LIN {X 0,Y 579.705,Z 783.31,A -85,B 0,C 180,E1 8978.544,E2 8978.544} C_VEL
LIN {X 0,Y 579.773,Z 783.31,A -85,B 0,C 180,E1 8983.301,E2 8983.301} C_VEL
LIN {X 0,Y 579.9,Z 783.31,A -85,B 0,C 180,E1 8989.468,E2 8989.468} C_VEL
LIN {X 0,Y 580.075,Z 783.31,A -85,B 0,C 180,E1 8994.009,E2 8994.009} C_VEL
LIN {X 0,Y 580.176,Z 783.31,A -85,B 0,C 180,E1 8998.509,E2 8998.509} C_VEL
LIN {X 0,Y 580.153,Z 783.31,A -85,B 0,C 180,E1 9002.999,E2 9002.999} C_VEL
LIN {X 0,Y 580.034,Z 783.31,A -85,B 0,C 180,E1 9007.51,E2 9007.51} C_VEL
LIN {X 0,Y 579.911,Z 783.31,A -85,B 0,C 180,E1 9012.07,E2 9012.07} C_VEL
LIN {X 0,Y 579.778,Z 783.31,A -85,B 0,C 180,E1 9016.711,E2 9016.711} C_VEL
LIN {X 0,Y 579.644,Z 783.31,A -85,B 0,C 180,E1 9021.47,E2 9021.47} C_VEL
LIN {X 0,Y 579.509,Z 783.31,A -85,B 0,C 180,E1 9027.261,E2 9027.261} C_VEL
LIN {X 0,Y 579.423,Z 783.31,A -85,B 0,C 180,E1 9033.311,E2 9033.311} C_VEL
LIN {X 0,Y 579.308,Z 783.31,A -85,B 0,C 180,E1 9038.885,E2 9038.885} C_VEL
LIN {X 0,Y 579.314,Z 783.31,A -85,B 0,C 180,E1 9045.078,E2 9045.078} C_VEL
LIN {X 0,Y 579.261,Z 783.31,A -85,B 0,C 180,E1 9051.116,E2 9051.116} C_VEL
LIN {X 0,Y 579.338,Z 783.519,A -85,B 0,C 180,E1 9053.514,E2 9053.514} C_VEL
LIN {X 0,Y 586.271,Z 797.884,A -85,B 0,C 180,E1 9054.256,E2 9054.256} C_VEL
LIN {X 0,Y 606.499,Z 837.506,A -85,B 0,C 180,E1 9056.265,E2 9056.265} C_VEL
LIN {X 0,Y 604.839,Z 881.39,A -85,B 0,C 180,E1 9057.125,E2 9057.125} C_VEL
LIN {X 0,Y 601.624,Z 924.158,A -85,B 0,C 180,E1 9058.57,E2 9058.57} C_VEL
LIN {X 0,Y 597.504,Z 964.209,A -85,B 0,C 180,E1 9060.574,E2 9060.574} C_VEL
LIN {X 0,Y 592.954,Z 1002,A -85,B 0,C 180,E1 9063.195,E2 9063.195} C_VEL
LIN {X 0,Y 588.505,Z 1036.812,A -85,B 0,C 180,E1 9066.46,E2 9066.46} C_VEL
LIN {X 0,Y 585.021,Z 1066.221,A -85,B 0,C 180,E1 9070.129,E2 9070.129} C_VEL
LIN {X 0,Y 582.678,Z 1089.161,A -85,B 0,C 180,E1 9073.891,E2 9073.891} C_VEL
LIN {X 0,Y 581.268,Z 1107.45,A -85,B 0,C 180,E1 9077.965,E2 9077.965} C_VEL
LIN {X 0,Y 580.663,Z 1119.244,A -85,B 0,C 180,E1 9081.75,E2 9081.75} C_VEL
LIN {X 0,Y 580.435,Z 1126.566,A -85,B 0,C 180,E1 9085.51,E2 9085.51} C_VEL
LIN {X 0,Y 580.498,Z 1129.543,A -85,B 0,C 180,E1 9090.001,E2 9090.001} C_VEL
LIN {X 0,Y 580.468,Z 1126.438,A -85,B 0,C 180,E1 9094.493,E2 9094.493} C_VEL
LIN {X 0,Y 580.72,Z 1119.016,A -85,B 0,C 180,E1 9098.252,E2 9098.252} C_VEL
LIN {X 0,Y 581.35,Z 1105.632,A -85,B 0,C 180,E1 9102.406,E2 9102.406} C_VEL
LIN {X 0,Y 582.795,Z 1087.275,A -85,B 0,C 180,E1 9106.362,E2 9106.362} C_VEL
LIN {X 0,Y 585.372,Z 1062.818,A -85,B 0,C 180,E1 9110.256,E2 9110.256} C_VEL
LIN {X 0,Y 588.867,Z 1034.215,A -85,B 0,C 180,E1 9113.721,E2 9113.721} C_VEL
LIN {X 0,Y 592.925,Z 1002.541,A -85,B 0,C 180,E1 9116.67,E2 9116.67} C_VEL
LIN {X 0,Y 597.544,Z 964.371,A -85,B 0,C 180,E1 9119.322,E2 9119.322} C_VEL
LIN {X 0,Y 601.491,Z 925.349,A -85,B 0,C 180,E1 9121.289,E2 9121.289} C_VEL
LIN {X 0,Y 604.713,Z 881.532,A -85,B 0,C 180,E1 9122.788,E2 9122.788} C_VEL
LIN {X 0,Y 606.403,Z 837.307,A -85,B 0,C 180,E1 9123.653,E2 9123.653} C_VEL
LIN {X 0,Y 579.444,Z 784.213,A -85,B 0,C 180,E1 9126.374,E2 9126.374} C_VEL
LIN {X 0,Y 579.393,Z 783.31,A -85,B 0,C 180,E1 9126.442,E2 9126.442} C_VEL
LIN {X 0,Y 579.354,Z 783.31,A -85,B 0,C 180,E1 9130.832,E2 9130.832} C_VEL
LIN {X 0,Y 579.285,Z 783.31,A -85,B 0,C 180,E1 9137.086,E2 9137.086} C_VEL
LIN {X 0,Y 579.266,Z 783.31,A -85,B 0,C 180,E1 9143.012,E2 9143.012} C_VEL
LIN {X 0,Y 579.458,Z 783.31,A -85,B 0,C 180,E1 9148.466,E2 9148.466} C_VEL
LIN {X 0,Y 579.564,Z 783.31,A -85,B 0,C 180,E1 9153.609,E2 9153.609} C_VEL
LIN {X 0,Y 579.673,Z 783.31,A -85,B 0,C 180,E1 9158.531,E2 9158.531} C_VEL
LIN {X 0,Y 579.784,Z 783.31,A -85,B 0,C 180,E1 9163.289,E2 9163.289} C_VEL
LIN {X 0,Y 579.956,Z 783.31,A -85,B 0,C 180,E1 9169.458,E2 9169.458} C_VEL
LIN {X 0,Y 580.11,Z 783.31,A -85,B 0,C 180,E1 9173.998,E2 9173.998} C_VEL
LIN {X 0,Y 580.202,Z 783.31,A -85,B 0,C 180,E1 9178.498,E2 9178.498} C_VEL
LIN {X 0,Y 580.166,Z 783.31,A -85,B 0,C 180,E1 9182.988,E2 9182.988} C_VEL
LIN {X 0,Y 580.046,Z 783.31,A -85,B 0,C 180,E1 9187.498,E2 9187.498} C_VEL
LIN {X 0,Y 579.912,Z 783.31,A -85,B 0,C 180,E1 9192.058,E2 9192.058} C_VEL
LIN {X 0,Y 579.821,Z 783.31,A -85,B 0,C 180,E1 9196.698,E2 9196.698} C_VEL
LIN {X 0,Y 579.67,Z 783.31,A -85,B 0,C 180,E1 9201.457,E2 9201.457} C_VEL
LIN {X 0,Y 579.573,Z 783.31,A -85,B 0,C 180,E1 9207.268,E2 9207.268} C_VEL
LIN {X 0,Y 579.449,Z 783.31,A -85,B 0,C 180,E1 9213.296,E2 9213.296} C_VEL
LIN {X 0,Y 579.272,Z 783.31,A -85,B 0,C 180,E1 9218.873,E2 9218.873} C_VEL
LIN {X 0,Y 579.22,Z 783.31,A -85,B 0,C 180,E1 9225.065,E2 9225.065} C_VEL
LIN {X 0,Y 579.372,Z 784.035,A -85,B 0,C 180,E1 9230.209,E2 9230.209} C_VEL
LIN {X 0,Y 603.342,Z 834.228,A -85,B 0,C 180,E1 9232.711,E2 9232.711} C_VEL
LIN {X 0,Y 607.455,Z 844.899,A -85,B 0,C 180,E1 9233.167,E2 9233.167} C_VEL
LIN {X 0,Y 605.623,Z 880.743,A -85,B 0,C 180,E1 9233.925,E2 9233.925} C_VEL
LIN {X 0,Y 600.996,Z 897.494,A -85,B 0,C 180,E1 9234.191,E2 9234.191} C_VEL
LIN {X 0,Y 596.819,Z 911.913,A -85,B 0,C 180,E1 9234.489,E2 9234.489} C_VEL
LIN {X 0,Y 596.616,Z 913.947,A -85,B 0,C 180,E1 9234.563,E2 9234.563} C_VEL
LIN {X 0,Y 592.607,Z 957.43,A -85,B 0,C 180,E1 9236.508,E2 9236.508} C_VEL
LIN {X 0,Y 588.124,Z 997.916,A -85,B 0,C 180,E1 9238.984,E2 9238.984} C_VEL
LIN {X 0,Y 583.838,Z 1034.56,A -85,B 0,C 180,E1 9241.907,E2 9241.907} C_VEL
LIN {X 0,Y 579.934,Z 1067.538,A -85,B 0,C 180,E1 9245.289,E2 9245.289} C_VEL
LIN {X 0,Y 576.663,Z 1096.856,A -85,B 0,C 180,E1 9249.175,E2 9249.175} C_VEL
LIN {X 0,Y 574.483,Z 1120.889,A -85,B 0,C 180,E1 9253.389,E2 9253.389} C_VEL
LIN {X 0,Y 573.307,Z 1137.76,A -85,B 0,C 180,E1 9257.405,E2 9257.405} C_VEL
LIN {X 0,Y 572.746,Z 1150.067,A -85,B 0,C 180,E1 9261.633,E2 9261.633} C_VEL
LIN {X 0,Y 572.529,Z 1156.644,A -85,B 0,C 180,E1 9265.445,E2 9265.445} C_VEL
LIN {X 0,Y 572.546,Z 1159.5,A -85,B 0,C 180,E1 9269.999,E2 9269.999} C_VEL
LIN {X 0,Y 572.544,Z 1156.648,A -85,B 0,C 180,E1 9274.552,E2 9274.552} C_VEL
LIN {X 0,Y 572.681,Z 1150.072,A -85,B 0,C 180,E1 9278.366,E2 9278.366} C_VEL
LIN {X 0,Y 573.309,Z 1137.771,A -85,B 0,C 180,E1 9282.592,E2 9282.592} C_VEL
LIN {X 0,Y 574.508,Z 1120.878,A -85,B 0,C 180,E1 9286.611,E2 9286.611} C_VEL
LIN {X 0,Y 576.684,Z 1096.833,A -85,B 0,C 180,E1 9290.827,E2 9290.827} C_VEL
LIN {X 0,Y 579.978,Z 1067.55,A -85,B 0,C 180,E1 9294.706,E2 9294.706} C_VEL
LIN {X 0,Y 583.804,Z 1034.632,A -85,B 0,C 180,E1 9298.087,E2 9298.087} C_VEL
LIN {X 0,Y 588.083,Z 997.958,A -85,B 0,C 180,E1 9301.015,E2 9301.015} C_VEL
LIN {X 0,Y 592.561,Z 957.205,A -85,B 0,C 180,E1 9303.507,E2 9303.507} C_VEL
LIN {X 0,Y 596.709,Z 912.308,A -85,B 0,C 180,E1 9305.503,E2 9305.503} C_VEL
LIN {X 0,Y 599.983,Z 864.038,A -85,B 0,C 180,E1 9306.907,E2 9306.907} C_VEL
LIN {X 0,Y 600.287,Z 844.634,A -85,B 0,C 180,E1 9307.314,E2 9307.314} C_VEL
LIN {X 0,Y 578.673,Z 798.345,A -85,B 0,C 180,E1 9309.62,E2 9309.62} C_VEL
LIN {X 0,Y 571.585,Z 784.671,A -85,B 0,C 180,E1 9310.396,E2 9310.396} C_VEL
LIN {X 0,Y 571.457,Z 783.31,A -85,B 0,C 180,E1 9310.504,E2 9310.504} C_VEL
LIN {X 0,Y 571.362,Z 783.31,A -85,B 0,C 180,E1 9316.424,E2 9316.424} C_VEL
LIN {X 0,Y 571.447,Z 783.31,A -85,B 0,C 180,E1 9322.694,E2 9322.694} C_VEL
LIN {X 0,Y 571.538,Z 783.31,A -85,B 0,C 180,E1 9328.028,E2 9328.028} C_VEL
LIN {X 0,Y 571.694,Z 783.31,A -85,B 0,C 180,E1 9333.23,E2 9333.23} C_VEL
LIN {X 0,Y 571.764,Z 783.31,A -85,B 0,C 180,E1 9338.231,E2 9338.231} C_VEL
LIN {X 0,Y 571.84,Z 783.31,A -85,B 0,C 180,E1 9343.062,E2 9343.062} C_VEL
LIN {X 0,Y 571.945,Z 783.31,A -85,B 0,C 180,E1 9348.567,E2 9348.567} C_VEL
LIN {X 0,Y 572.179,Z 783.31,A -85,B 0,C 180,E1 9353.926,E2 9353.926} C_VEL
LIN {X 0,Y 572.274,Z 783.31,A -85,B 0,C 180,E1 9358.489,E2 9358.489} C_VEL
LIN {X 0,Y 572.253,Z 783.31,A -85,B 0,C 180,E1 9363.041,E2 9363.041} C_VEL
LIN {X 0,Y 572.117,Z 783.31,A -85,B 0,C 180,E1 9367.614,E2 9367.614} C_VEL
LIN {X 0,Y 572.013,Z 783.31,A -85,B 0,C 180,E1 9372.239,E2 9372.239} C_VEL
LIN {X 0,Y 571.803,Z 783.31,A -85,B 0,C 180,E1 9377.464,E2 9377.464} C_VEL
LIN {X 0,Y 571.684,Z 783.31,A -85,B 0,C 180,E1 9383.429,E2 9383.429} C_VEL
LIN {X 0,Y 571.542,Z 783.31,A -85,B 0,C 180,E1 9388.978,E2 9388.978} C_VEL
LIN {X 0,Y 571.413,Z 783.31,A -85,B 0,C 180,E1 9394.717,E2 9394.717} C_VEL
LIN {X 0,Y 571.347,Z 783.31,A -85,B 0,C 180,E1 9399.733,E2 9399.733} C_VEL
LIN {X 0,Y 571.329,Z 783.31,A -85,B 0,C 180,E1 9405.731,E2 9405.731} C_VEL
LIN {X 0,Y 571.304,Z 783.31,A -85,B 0,C 180,E1 9410.47,E2 9410.47} C_VEL
LIN {X 0,Y 571.377,Z 783.363,A -85,B 0,C 180,E1 9412.878,E2 9412.878} C_VEL
LIN {X 0,Y 575.876,Z 793.256,A -85,B 0,C 180,E1 9413.386,E2 9413.386} C_VEL
LIN {X 0,Y 599.985,Z 840.052,A -85,B 0,C 180,E1 9415.857,E2 9415.857} C_VEL
LIN {X 0,Y 598.239,Z 883.352,A -85,B 0,C 180,E1 9416.746,E2 9416.746} C_VEL
LIN {X 0,Y 594.976,Z 924.317,A -85,B 0,C 180,E1 9418.148,E2 9418.148} C_VEL
LIN {X 0,Y 590.642,Z 964.871,A -85,B 0,C 180,E1 9420.198,E2 9420.198} C_VEL
LIN {X 0,Y 585.854,Z 1002.667,A -85,B 0,C 180,E1 9422.847,E2 9422.847} C_VEL
LIN {X 0,Y 581.235,Z 1037.328,A -85,B 0,C 180,E1 9426.134,E2 9426.134} C_VEL
LIN {X 0,Y 577.487,Z 1066.722,A -85,B 0,C 180,E1 9429.858,E2 9429.858} C_VEL
LIN {X 0,Y 574.912,Z 1090.243,A -85,B 0,C 180,E1 9433.81,E2 9433.81} C_VEL
LIN {X 0,Y 573.435,Z 1108.002,A -85,B 0,C 180,E1 9437.862,E2 9437.862} C_VEL
LIN {X 0,Y 572.791,Z 1119.491,A -85,B 0,C 180,E1 9441.636,E2 9441.636} C_VEL
LIN {X 0,Y 572.549,Z 1126.783,A -85,B 0,C 180,E1 9445.448,E2 9445.448} C_VEL
LIN {X 0,Y 572.624,Z 1129.751,A -85,B 0,C 180,E1 9450.001,E2 9450.001} C_VEL
LIN {X 0,Y 572.577,Z 1126.658,A -85,B 0,C 180,E1 9454.555,E2 9454.555} C_VEL
LIN {X 0,Y 572.836,Z 1119.262,A -85,B 0,C 180,E1 9458.366,E2 9458.366} C_VEL
LIN {X 0,Y 573.562,Z 1105.901,A -85,B 0,C 180,E1 9462.589,E2 9462.589} C_VEL
LIN {X 0,Y 575.106,Z 1087.461,A -85,B 0,C 180,E1 9466.627,E2 9466.627} C_VEL
LIN {X 0,Y 577.863,Z 1063.364,A -85,B 0,C 180,E1 9470.531,E2 9470.531} C_VEL
LIN {X 0,Y 581.7,Z 1034.06,A -85,B 0,C 180,E1 9474.123,E2 9474.123} C_VEL
LIN {X 0,Y 586.115,Z 1001.197,A -85,B 0,C 180,E1 9477.172,E2 9477.172} C_VEL
LIN {X 0,Y 590.67,Z 965.045,A -85,B 0,C 180,E1 9479.697,E2 9479.697} C_VEL
LIN {X 0,Y 594.908,Z 924.983,A -85,B 0,C 180,E1 9481.732,E2 9481.732} C_VEL
LIN {X 0,Y 598.217,Z 881.836,A -85,B 0,C 180,E1 9483.215,E2 9483.215} C_VEL
LIN {X 0,Y 599.71,Z 839.363,A -85,B 0,C 180,E1 9484.081,E2 9484.081} C_VEL
LIN {X 0,Y 573.027,Z 788.001,A -85,B 0,C 180,E1 9486.825,E2 9486.825} C_VEL
LIN {X 0,Y 571.451,Z 783.31,A -85,B 0,C 180,E1 9487.076,E2 9487.076} C_VEL
LIN {X 0,Y 571.368,Z 783.31,A -85,B 0,C 180,E1 9492.052,E2 9492.052} C_VEL
LIN {X 0,Y 571.326,Z 783.31,A -85,B 0,C 180,E1 9497.952,E2 9497.952} C_VEL
LIN {X 0,Y 571.374,Z 783.31,A -85,B 0,C 180,E1 9504.307,E2 9504.307} C_VEL
LIN {X 0,Y 571.546,Z 783.31,A -85,B 0,C 180,E1 9509.752,E2 9509.752} C_VEL
LIN {X 0,Y 571.651,Z 783.31,A -85,B 0,C 180,E1 9514.904,E2 9514.904} C_VEL
LIN {X 0,Y 571.792,Z 783.31,A -85,B 0,C 180,E1 9519.846,E2 9519.846} C_VEL
LIN {X 0,Y 571.886,Z 783.31,A -85,B 0,C 180,E1 9524.632,E2 9524.632} C_VEL
LIN {X 0,Y 572.032,Z 783.31,A -85,B 0,C 180,E1 9529.31,E2 9529.31} C_VEL
LIN {X 0,Y 572.215,Z 783.31,A -85,B 0,C 180,E1 9533.915,E2 9533.915} C_VEL
LIN {X 0,Y 572.3,Z 783.31,A -85,B 0,C 180,E1 9538.477,E2 9538.477} C_VEL
LIN {X 0,Y 572.266,Z 783.31,A -85,B 0,C 180,E1 9543.029,E2 9543.029} C_VEL
LIN {X 0,Y 572.129,Z 783.31,A -85,B 0,C 180,E1 9547.603,E2 9547.603} C_VEL
LIN {X 0,Y 572.016,Z 783.31,A -85,B 0,C 180,E1 9552.227,E2 9552.227} C_VEL
LIN {X 0,Y 571.861,Z 783.31,A -85,B 0,C 180,E1 9557.474,E2 9557.474} C_VEL
LIN {X 0,Y 571.713,Z 783.31,A -85,B 0,C 180,E1 9563.416,E2 9563.416} C_VEL
LIN {X 0,Y 571.606,Z 783.31,A -85,B 0,C 180,E1 9568.984,E2 9568.984} C_VEL
LIN {X 0,Y 571.441,Z 783.31,A -85,B 0,C 180,E1 9574.716,E2 9574.716} C_VEL
LIN {X 0,Y 571.307,Z 783.31,A -85,B 0,C 180,E1 9579.724,E2 9579.724} C_VEL
LIN {X 0,Y 571.244,Z 783.31,A -85,B 0,C 180,E1 9585.724,E2 9585.724} C_VEL
LIN {X 0,Y 571.386,Z 783.31,A -85,B 0,C 180,E1 9589.55,E2 9589.55} C_VEL
LIN {X 0,Y 578.3,Z 797.9,A -85,B 0,C 180,E1 9590.349,E2 9590.349} C_VEL
LIN {X 0,Y 597.471,Z 838.23,A -85,B 0,C 180,E1 9592.384,E2 9592.384} C_VEL
LIN {X 0,Y 600.887,Z 848.155,A -85,B 0,C 180,E1 9592.792,E2 9592.792} C_VEL
LIN {X 0,Y 597.909,Z 896.617,A -85,B 0,C 180,E1 9593.962,E2 9593.962} C_VEL
LIN {X 0,Y 596.616,Z 913.947,A -85,B 0,C 180,E1 9594.563,E2 9594.563} C_VEL
LIN {X 0,Y 591.957,Z 930.184,A -85,B 0,C 180,E1 9595.009,E2 9595.009} C_VEL
LIN {X 0,Y 586.881,Z 946.086,A -85,B 0,C 180,E1 9595.525,E2 9595.525} C_VEL
LIN {X 0,Y 582.246,Z 987.803,A -85,B 0,C 180,E1 9597.91,E2 9597.91} C_VEL
LIN {X 0,Y 577.374,Z 1027.62,A -85,B 0,C 180,E1 9600.954,E2 9600.954} C_VEL
LIN {X 0,Y 572.843,Z 1063.537,A -85,B 0,C 180,E1 9604.539,E2 9604.539} C_VEL
LIN {X 0,Y 569.357,Z 1093.631,A -85,B 0,C 180,E1 9608.469,E2 9608.469} C_VEL
LIN {X 0,Y 566.949,Z 1117.235,A -85,B 0,C 180,E1 9612.502,E2 9612.502} C_VEL
LIN {X 0,Y 565.582,Z 1134.682,A -85,B 0,C 180,E1 9616.442,E2 9616.442} C_VEL
LIN {X 0,Y 564.92,Z 1148.033,A -85,B 0,C 180,E1 9620.738,E2 9620.738} C_VEL
LIN {X 0,Y 564.774,Z 1155.665,A -85,B 0,C 180,E1 9624.611,E2 9624.611} C_VEL
LIN {X 0,Y 564.576,Z 1159.164,A -85,B 0,C 180,E1 9628.461,E2 9628.461} C_VEL
LIN {X 0,Y 564.671,Z 1158.213,A -85,B 0,C 180,E1 9633.075,E2 9633.075} C_VEL
LIN {X 0,Y 564.718,Z 1153.025,A -85,B 0,C 180,E1 9637.006,E2 9637.006} C_VEL
LIN {X 0,Y 565.2,Z 1141.864,A -85,B 0,C 180,E1 9641.461,E2 9641.461} C_VEL
LIN {X 0,Y 566.303,Z 1126.073,A -85,B 0,C 180,E1 9645.634,E2 9645.634} C_VEL
LIN {X 0,Y 568.3,Z 1104.157,A -85,B 0,C 180,E1 9649.871,E2 9649.871} C_VEL
LIN {X 0,Y 571.506,Z 1075.51,A -85,B 0,C 180,E1 9654.023,E2 9654.023} C_VEL
LIN {X 0,Y 575.713,Z 1040.738,A -85,B 0,C 180,E1 9657.848,E2 9657.848} C_VEL
LIN {X 0,Y 580.574,Z 1001.704,A -85,B 0,C 180,E1 9661.123,E2 9661.123} C_VEL
LIN {X 0,Y 585.507,Z 959.146,A -85,B 0,C 180,E1 9663.809,E2 9663.809} C_VEL
LIN {X 0,Y 589.994,Z 913.311,A -85,B 0,C 180,E1 9665.888,E2 9665.888} C_VEL
LIN {X 0,Y 593.477,Z 864.388,A -85,B 0,C 180,E1 9667.336,E2 9667.336} C_VEL
LIN {X 0,Y 593.69,Z 847.037,A -85,B 0,C 180,E1 9667.722,E2 9667.722} C_VEL
LIN {X 0,Y 573.213,Z 802.88,A -85,B 0,C 180,E1 9669.97,E2 9669.97} C_VEL
LIN {X 0,Y 563.625,Z 784.43,A -85,B 0,C 180,E1 9671.049,E2 9671.049} C_VEL
LIN {X 0,Y 563.53,Z 783.31,A -85,B 0,C 180,E1 9671.178,E2 9671.178} C_VEL
LIN {X 0,Y 563.45,Z 783.31,A -85,B 0,C 180,E1 9676.554,E2 9676.554} C_VEL
LIN {X 0,Y 563.427,Z 783.31,A -85,B 0,C 180,E1 9681.804,E2 9681.804} C_VEL
LIN {X 0,Y 563.547,Z 783.31,A -85,B 0,C 180,E1 9687.481,E2 9687.481} C_VEL
LIN {X 0,Y 563.726,Z 783.31,A -85,B 0,C 180,E1 9692.821,E2 9692.821} C_VEL
LIN {X 0,Y 563.856,Z 783.31,A -85,B 0,C 180,E1 9697.91,E2 9697.91} C_VEL
LIN {X 0,Y 563.946,Z 783.31,A -85,B 0,C 180,E1 9702.818,E2 9702.818} C_VEL
LIN {X 0,Y 564.001,Z 783.31,A -85,B 0,C 180,E1 9707.596,E2 9707.596} C_VEL
LIN {X 0,Y 564.253,Z 783.31,A -85,B 0,C 180,E1 9713.474,E2 9713.474} C_VEL
LIN {X 0,Y 564.372,Z 783.31,A -85,B 0,C 180,E1 9718.468,E2 9718.468} C_VEL
LIN {X 0,Y 564.349,Z 783.31,A -85,B 0,C 180,E1 9723.084,E2 9723.084} C_VEL
LIN {X 0,Y 564.215,Z 783.31,A -85,B 0,C 180,E1 9727.722,E2 9727.722} C_VEL
LIN {X 0,Y 564.085,Z 783.31,A -85,B 0,C 180,E1 9732.413,E2 9732.413} C_VEL
LIN {X 0,Y 563.939,Z 783.31,A -85,B 0,C 180,E1 9737.194,E2 9737.194} C_VEL
LIN {X 0,Y 563.793,Z 783.31,A -85,B 0,C 180,E1 9742.105,E2 9742.105} C_VEL
LIN {X 0,Y 563.621,Z 783.31,A -85,B 0,C 180,E1 9747.489,E2 9747.489} C_VEL
LIN {X 0,Y 563.528,Z 783.31,A -85,B 0,C 180,E1 9752.533,E2 9752.533} C_VEL
LIN {X 0,Y 563.418,Z 783.31,A -85,B 0,C 180,E1 9758.212,E2 9758.212} C_VEL
LIN {X 0,Y 563.447,Z 783.31,A -85,B 0,C 180,E1 9763.445,E2 9763.445} C_VEL
LIN {X 0,Y 563.39,Z 783.31,A -85,B 0,C 180,E1 9768.856,E2 9768.856} C_VEL
LIN {X 0,Y 563.417,Z 783.31,A -85,B 0,C 180,E1 9772.213,E2 9772.213} C_VEL
LIN {X 0,Y 567.985,Z 793.236,A -85,B 0,C 180,E1 9772.751,E2 9772.751} C_VEL
LIN {X 0,Y 593.65,Z 842.846,A -85,B 0,C 180,E1 9775.457,E2 9775.457} C_VEL
LIN {X 0,Y 591.703,Z 884.356,A -85,B 0,C 180,E1 9776.33,E2 9776.33} C_VEL
LIN {X 0,Y 588.228,Z 925.883,A -85,B 0,C 180,E1 9777.782,E2 9777.782} C_VEL
LIN {X 0,Y 583.764,Z 965.464,A -85,B 0,C 180,E1 9779.811,E2 9779.811} C_VEL
LIN {X 0,Y 578.862,Z 1002.511,A -85,B 0,C 180,E1 9782.432,E2 9782.432} C_VEL
LIN {X 0,Y 574.009,Z 1037.146,A -85,B 0,C 180,E1 9785.731,E2 9785.731} C_VEL
LIN {X 0,Y 570.172,Z 1065.958,A -85,B 0,C 180,E1 9789.388,E2 9789.388} C_VEL
LIN {X 0,Y 567.403,Z 1089.086,A -85,B 0,C 180,E1 9793.281,E2 9793.281} C_VEL
LIN {X 0,Y 565.661,Z 1108.061,A -85,B 0,C 180,E1 9797.628,E2 9797.628} C_VEL
LIN {X 0,Y 564.947,Z 1119.74,A -85,B 0,C 180,E1 9801.519,E2 9801.519} C_VEL
LIN {X 0,Y 564.658,Z 1127,A -85,B 0,C 180,E1 9805.384,E2 9805.384} C_VEL
LIN {X 0,Y 564.725,Z 1129.96,A -85,B 0,C 180,E1 9810.001,E2 9810.001} C_VEL
LIN {X 0,Y 564.683,Z 1126.88,A -85,B 0,C 180,E1 9814.618,E2 9814.618} C_VEL
LIN {X 0,Y 564.977,Z 1119.52,A -85,B 0,C 180,E1 9818.483,E2 9818.483} C_VEL
LIN {X 0,Y 565.748,Z 1106.214,A -85,B 0,C 180,E1 9822.766,E2 9822.766} C_VEL
LIN {X 0,Y 567.366,Z 1088.608,A -85,B 0,C 180,E1 9826.723,E2 9826.723} C_VEL
LIN {X 0,Y 570.345,Z 1063.906,A -85,B 0,C 180,E1 9830.814,E2 9830.814} C_VEL
LIN {X 0,Y 574.393,Z 1034.59,A -85,B 0,C 180,E1 9834.449,E2 9834.449} C_VEL
LIN {X 0,Y 579.113,Z 1001.162,A -85,B 0,C 180,E1 9837.578,E2 9837.578} C_VEL
LIN {X 0,Y 583.994,Z 964.006,A -85,B 0,C 180,E1 9840.179,E2 9840.179} C_VEL
LIN {X 0,Y 588.317,Z 925.016,A -85,B 0,C 180,E1 9842.165,E2 9842.165} C_VEL
LIN {X 0,Y 591.847,Z 881.288,A -85,B 0,C 180,E1 9843.672,E2 9843.672} C_VEL
LIN {X 0,Y 593.299,Z 842.018,A -85,B 0,C 180,E1 9844.49,E2 9844.49} C_VEL
LIN {X 0,Y 565.406,Z 788.412,A -85,B 0,C 180,E1 9847.439,E2 9847.439} C_VEL
LIN {X 0,Y 563.511,Z 783.31,A -85,B 0,C 180,E1 9847.731,E2 9847.731} C_VEL
LIN {X 0,Y 563.458,Z 783.31,A -85,B 0,C 180,E1 9853.442,E2 9853.442} C_VEL
LIN {X 0,Y 563.392,Z 783.31,A -85,B 0,C 180,E1 9858.855,E2 9858.855} C_VEL
LIN {X 0,Y 563.436,Z 783.31,A -85,B 0,C 180,E1 9863.781,E2 9863.781} C_VEL
LIN {X 0,Y 563.625,Z 783.31,A -85,B 0,C 180,E1 9869.346,E2 9869.346} C_VEL
LIN {X 0,Y 563.728,Z 783.31,A -85,B 0,C 180,E1 9874.526,E2 9874.526} C_VEL
LIN {X 0,Y 563.874,Z 783.31,A -85,B 0,C 180,E1 9880.134,E2 9880.134} C_VEL
LIN {X 0,Y 563.976,Z 783.31,A -85,B 0,C 180,E1 9886.003,E2 9886.003} C_VEL
LIN {X 0,Y 564.173,Z 783.31,A -85,B 0,C 180,E1 9890.722,E2 9890.722} C_VEL
LIN {X 0,Y 564.352,Z 783.31,A -85,B 0,C 180,E1 9895.375,E2 9895.375} C_VEL
LIN {X 0,Y 564.531,Z 783.31,A -85,B 0,C 180,E1 9901.532,E2 9901.532} C_VEL
LIN {X 0,Y 564.278,Z 783.31,A -85,B 0,C 180,E1 9906.526,E2 9906.526} C_VEL
LIN {X 0,Y 564.091,Z 783.31,A -85,B 0,C 180,E1 9912.402,E2 9912.402} C_VEL
LIN {X 0,Y 563.987,Z 783.31,A -85,B 0,C 180,E1 9917.181,E2 9917.181} C_VEL
LIN {X 0,Y 563.818,Z 783.31,A -85,B 0,C 180,E1 9922.092,E2 9922.092} C_VEL
LIN {X 0,Y 563.686,Z 783.31,A -85,B 0,C 180,E1 9927.495,E2 9927.495} C_VEL
LIN {X 0,Y 563.576,Z 783.31,A -85,B 0,C 180,E1 9932.517,E2 9932.517} C_VEL
LIN {X 0,Y 563.39,Z 783.31,A -85,B 0,C 180,E1 9938.199,E2 9938.199} C_VEL
LIN {X 0,Y 563.355,Z 783.31,A -85,B 0,C 180,E1 9943.432,E2 9943.432} C_VEL
LIN {X 0,Y 563.431,Z 783.31,A -85,B 0,C 180,E1 9948.9,E2 9948.9} C_VEL
LIN {X 0,Y 570.232,Z 797.568,A -85,B 0,C 180,E1 9949.713,E2 9949.713} C_VEL
LIN {X 0,Y 588.981,Z 835.971,A -85,B 0,C 180,E1 9951.749,E2 9951.749} C_VEL
LIN {X 0,Y 594.335,Z 850.339,A -85,B 0,C 180,E1 9952.397,E2 9952.397} C_VEL
LIN {X 0,Y 591.262,Z 897.439,A -85,B 0,C 180,E1 9953.561,E2 9953.561} C_VEL
LIN {X 0,Y 587.286,Z 941.765,A -85,B 0,C 180,E1 9955.314,E2 9955.314} C_VEL
LIN {X 0,Y 586.881,Z 946.086,A -85,B 0,C 180,E1 9955.525,E2 9955.525} C_VEL
LIN {X 0,Y 581.755,Z 961.748,A -85,B 0,C 180,E1 9956.133,E2 9956.133} C_VEL
LIN {X 0,Y 576.59,Z 976.908,A -85,B 0,C 180,E1 9956.821,E2 9956.821} C_VEL
LIN {X 0,Y 571.558,Z 1016.512,A -85,B 0,C 180,E1 9959.655,E2 9959.655} C_VEL
LIN {X 0,Y 566.708,Z 1053.571,A -85,B 0,C 180,E1 9963.139,E2 9963.139} C_VEL
LIN {X 0,Y 562.713,Z 1085.318,A -85,B 0,C 180,E1 9967.017,E2 9967.017} C_VEL
LIN {X 0,Y 559.69,Z 1112.051,A -85,B 0,C 180,E1 9971.318,E2 9971.318} C_VEL
LIN {X 0,Y 557.998,Z 1131.258,A -85,B 0,C 180,E1 9975.457,E2 9975.457} C_VEL
LIN {X 0,Y 557.148,Z 1145.807,A -85,B 0,C 180,E1 9979.817,E2 9979.817} C_VEL
LIN {X 0,Y 556.874,Z 1155.46,A -85,B 0,C 180,E1 9984.534,E2 9984.534} C_VEL
LIN {X 0,Y 556.674,Z 1159.029,A -85,B 0,C 180,E1 9988.439,E2 9988.439} C_VEL
LIN {X 0,Y 556.653,Z 1159.029,A -85,B 0,C 180,E1 9991.558,E2 9991.558} C_VEL
LIN {X 0,Y 556.839,Z 1154.228,A -85,B 0,C 180,E1 9996.247,E2 9996.247} C_VEL
LIN {X 0,Y 557.152,Z 1144.698,A -85,B 0,C 180,E1 10000.576,E2 10000.576} C_VEL
LIN {X 0,Y 558.171,Z 1129.681,A -85,B 0,C 180,E1 10004.937,E2 10004.937} C_VEL
LIN {X 0,Y 559.934,Z 1109.417,A -85,B 0,C 180,E1 10009.152,E2 10009.152} C_VEL
LIN {X 0,Y 562.858,Z 1083.827,A -85,B 0,C 180,E1 10013.183,E2 10013.183} C_VEL
LIN {X 0,Y 566.851,Z 1052.043,A -85,B 0,C 180,E1 10017.025,E2 10017.025} C_VEL
LIN {X 0,Y 571.821,Z 1014.353,A -85,B 0,C 180,E1 10020.525,E2 10020.525} C_VEL
LIN {X 0,Y 577.051,Z 973.564,A -85,B 0,C 180,E1 10023.391,E2 10023.391} C_VEL
LIN {X 0,Y 581.831,Z 929.692,A -85,B 0,C 180,E1 10025.658,E2 10025.658} C_VEL
LIN {X 0,Y 585.764,Z 885.326,A -85,B 0,C 180,E1 10027.234,E2 10027.234} C_VEL
LIN {X 0,Y 587.285,Z 849.917,A -85,B 0,C 180,E1 10028.109,E2 10028.109} C_VEL
LIN {X 0,Y 568.195,Z 808.203,A -85,B 0,C 180,E1 10030.281,E2 10030.281} C_VEL
LIN {X 0,Y 555.618,Z 784.03,A -85,B 0,C 180,E1 10031.734,E2 10031.734} C_VEL
LIN {X 0,Y 555.535,Z 783.31,A -85,B 0,C 180,E1 10037.423,E2 10037.423} C_VEL
LIN {X 0,Y 555.499,Z 783.31,A -85,B 0,C 180,E1 10043.137,E2 10043.137} C_VEL
LIN {X 0,Y 555.669,Z 783.31,A -85,B 0,C 180,E1 10048.807,E2 10048.807} C_VEL
LIN {X 0,Y 555.856,Z 783.31,A -85,B 0,C 180,E1 10054.152,E2 10054.152} C_VEL
LIN {X 0,Y 555.926,Z 783.31,A -85,B 0,C 180,E1 10059.257,E2 10059.257} C_VEL
LIN {X 0,Y 556.018,Z 783.31,A -85,B 0,C 180,E1 10064.194,E2 10064.194} C_VEL
LIN {X 0,Y 556.158,Z 783.31,A -85,B 0,C 180,E1 10069.013,E2 10069.013} C_VEL
LIN {X 0,Y 556.378,Z 783.31,A -85,B 0,C 180,E1 10073.753,E2 10073.753} C_VEL
LIN {X 0,Y 556.476,Z 783.31,A -85,B 0,C 180,E1 10078.446,E2 10078.446} C_VEL
LIN {X 0,Y 556.454,Z 783.31,A -85,B 0,C 180,E1 10083.127,E2 10083.127} C_VEL
LIN {X 0,Y 556.295,Z 783.31,A -85,B 0,C 180,E1 10087.832,E2 10087.832} C_VEL
LIN {X 0,Y 556.181,Z 783.31,A -85,B 0,C 180,E1 10092.593,E2 10092.593} C_VEL
LIN {X 0,Y 555.996,Z 783.31,A -85,B 0,C 180,E1 10097.49,E2 10097.49} C_VEL
LIN {X 0,Y 555.866,Z 783.31,A -85,B 0,C 180,E1 10102.437,E2 10102.437} C_VEL
LIN {X 0,Y 555.716,Z 783.31,A -85,B 0,C 180,E1 10107.617,E2 10107.617} C_VEL
LIN {X 0,Y 555.617,Z 783.31,A -85,B 0,C 180,E1 10113.055,E2 10113.055} C_VEL
LIN {X 0,Y 555.522,Z 783.31,A -85,B 0,C 180,E1 10118.856,E2 10118.856} C_VEL
LIN {X 0,Y 555.513,Z 783.31,A -85,B 0,C 180,E1 10124.836,E2 10124.836} C_VEL
LIN {X 0,Y 555.478,Z 783.31,A -85,B 0,C 180,E1 10129.799,E2 10129.799} C_VEL
LIN {X 0,Y 555.468,Z 783.31,A -85,B 0,C 180,E1 10131.533,E2 10131.533} C_VEL
LIN {X 0,Y 559.757,Z 792.791,A -85,B 0,C 180,E1 10132.058,E2 10132.058} C_VEL
LIN {X 0,Y 587.275,Z 845.51,A -85,B 0,C 180,E1 10135.041,E2 10135.041} C_VEL
LIN {X 0,Y 585.188,Z 885.344,A -85,B 0,C 180,E1 10135.904,E2 10135.904} C_VEL
LIN {X 0,Y 581.649,Z 925.679,A -85,B 0,C 180,E1 10137.327,E2 10137.327} C_VEL
LIN {X 0,Y 576.926,Z 965.996,A -85,B 0,C 180,E1 10139.415,E2 10139.415} C_VEL
LIN {X 0,Y 571.691,Z 1003.818,A -85,B 0,C 180,E1 10142.134,E2 10142.134} C_VEL
LIN {X 0,Y 566.813,Z 1037.144,A -85,B 0,C 180,E1 10145.351,E2 10145.351} C_VEL
LIN {X 0,Y 562.593,Z 1066.693,A -85,B 0,C 180,E1 10149.144,E2 10149.144} C_VEL
LIN {X 0,Y 559.741,Z 1089.704,A -85,B 0,C 180,E1 10153.084,E2 10153.084} C_VEL
LIN {X 0,Y 557.856,Z 1108.38,A -85,B 0,C 180,E1 10157.452,E2 10157.452} C_VEL
LIN {X 0,Y 557.088,Z 1119.995,A -85,B 0,C 180,E1 10161.398,E2 10161.398} C_VEL
LIN {X 0,Y 556.768,Z 1127.219,A -85,B 0,C 180,E1 10165.318,E2 10165.318} C_VEL
LIN {X 0,Y 556.827,Z 1130.167,A -85,B 0,C 180,E1 10170.001,E2 10170.001} C_VEL
LIN {X 0,Y 556.791,Z 1127.104,A -85,B 0,C 180,E1 10174.684,E2 10174.684} C_VEL
LIN {X 0,Y 557.11,Z 1119.774,A -85,B 0,C 180,E1 10178.604,E2 10178.604} C_VEL
LIN {X 0,Y 557.946,Z 1106.549,A -85,B 0,C 180,E1 10182.948,E2 10182.948} C_VEL
LIN {X 0,Y 559.772,Z 1088.183,A -85,B 0,C 180,E1 10187.12,E2 10187.12} C_VEL
LIN {X 0,Y 562.797,Z 1064.745,A -85,B 0,C 180,E1 10191.052,E2 10191.052} C_VEL
LIN {X 0,Y 567.006,Z 1035.91,A -85,B 0,C 180,E1 10194.692,E2 10194.692} C_VEL
LIN {X 0,Y 571.952,Z 1002.439,A -85,B 0,C 180,E1 10197.886,E2 10197.886} C_VEL
LIN {X 0,Y 577.17,Z 964.591,A -85,B 0,C 180,E1 10200.574,E2 10200.574} C_VEL
LIN {X 0,Y 581.72,Z 925.39,A -85,B 0,C 180,E1 10202.591,E2 10202.591} C_VEL
LIN {X 0,Y 585.415,Z 881.472,A -85,B 0,C 180,E1 10204.12,E2 10204.12} C_VEL
LIN {X 0,Y 586.747,Z 844.389,A -85,B 0,C 180,E1 10204.924,E2 10204.924} C_VEL
LIN {X 0,Y 560.262,Z 793.41,A -85,B 0,C 180,E1 10207.793,E2 10207.793} C_VEL
LIN {X 0,Y 555.541,Z 783.31,A -85,B 0,C 180,E1 10208.413,E2 10208.413} C_VEL
LIN {X 0,Y 555.534,Z 783.31,A -85,B 0,C 180,E1 10212.99,E2 10212.99} C_VEL
LIN {X 0,Y 555.488,Z 783.31,A -85,B 0,C 180,E1 10219.105,E2 10219.105} C_VEL
LIN {X 0,Y 555.494,Z 783.31,A -85,B 0,C 180,E1 10225.051,E2 10225.051} C_VEL
LIN {X 0,Y 555.748,Z 783.31,A -85,B 0,C 180,E1 10230.745,E2 10230.745} C_VEL
LIN {X 0,Y 555.834,Z 783.31,A -85,B 0,C 180,E1 10235.861,E2 10235.861} C_VEL
LIN {X 0,Y 556.004,Z 783.31,A -85,B 0,C 180,E1 10240.908,E2 10240.908} C_VEL
LIN {X 0,Y 556.074,Z 783.31,A -85,B 0,C 180,E1 10245.8,E2 10245.8} C_VEL
LIN {X 0,Y 556.253,Z 783.31,A -85,B 0,C 180,E1 10250.589,E2 10250.589} C_VEL
LIN {X 0,Y 556.446,Z 783.31,A -85,B 0,C 180,E1 10255.309,E2 10255.309} C_VEL
LIN {X 0,Y 556.624,Z 783.31,A -85,B 0,C 180,E1 10261.554,E2 10261.554} C_VEL
LIN {X 0,Y 556.408,Z 783.31,A -85,B 0,C 180,E1 10266.247,E2 10266.247} C_VEL
LIN {X 0,Y 556.188,Z 783.31,A -85,B 0,C 180,E1 10272.581,E2 10272.581} C_VEL
LIN {X 0,Y 556.069,Z 783.31,A -85,B 0,C 180,E1 10277.504,E2 10277.504} C_VEL
LIN {X 0,Y 555.885,Z 783.31,A -85,B 0,C 180,E1 10282.424,E2 10282.424} C_VEL
LIN {X 0,Y 555.804,Z 783.31,A -85,B 0,C 180,E1 10287.599,E2 10287.599} C_VEL
LIN {X 0,Y 555.651,Z 783.31,A -85,B 0,C 180,E1 10293.039,E2 10293.039} C_VEL
LIN {X 0,Y 555.487,Z 783.31,A -85,B 0,C 180,E1 10298.843,E2 10298.843} C_VEL
LIN {X 0,Y 555.427,Z 783.31,A -85,B 0,C 180,E1 10304.823,E2 10304.823} C_VEL
LIN {X 0,Y 555.51,Z 783.757,A -85,B 0,C 180,E1 10308.26,E2 10308.26} C_VEL
LIN {X 0,Y 581.481,Z 835.926,A -85,B 0,C 180,E1 10311.204,E2 10311.204} C_VEL
LIN {X 0,Y 587.805,Z 852.1,A -85,B 0,C 180,E1 10311.982,E2 10311.982} C_VEL
LIN {X 0,Y 584.654,Z 898.165,A -85,B 0,C 180,E1 10313.147,E2 10313.147} C_VEL
LIN {X 0,Y 580.458,Z 943.013,A -85,B 0,C 180,E1 10314.95,E2 10314.95} C_VEL
LIN {X 0,Y 576.59,Z 976.908,A -85,B 0,C 180,E1 10316.821,E2 10316.821} C_VEL
LIN {X 0,Y 571.318,Z 991.763,A -85,B 0,C 180,E1 10317.599,E2 10317.599} C_VEL
LIN {X 0,Y 565.886,Z 1006.093,A -85,B 0,C 180,E1 10318.449,E2 10318.449} C_VEL
LIN {X 0,Y 560.929,Z 1041.756,A -85,B 0,C 180,E1 10321.579,E2 10321.579} C_VEL
LIN {X 0,Y 556.293,Z 1075.753,A -85,B 0,C 180,E1 10325.457,E2 10325.457} C_VEL
LIN {X 0,Y 552.827,Z 1104.518,A -85,B 0,C 180,E1 10329.754,E2 10329.754} C_VEL
LIN {X 0,Y 550.509,Z 1127.513,A -85,B 0,C 180,E1 10334.389,E2 10334.389} C_VEL
LIN {X 0,Y 549.403,Z 1143.258,A -85,B 0,C 180,E1 10338.868,E2 10338.868} C_VEL
LIN {X 0,Y 548.943,Z 1152.854,A -85,B 0,C 180,E1 10342.943,E2 10342.943} C_VEL
LIN {X 0,Y 548.802,Z 1157.847,A -85,B 0,C 180,E1 10346.833,E2 10346.833} C_VEL
LIN {X 0,Y 548.848,Z 1159.165,A -85,B 0,C 180,E1 10349.999,E2 10349.999} C_VEL
LIN {X 0,Y 548.866,Z 1156.242,A -85,B 0,C 180,E1 10354.749,E2 10354.749} C_VEL
LIN {X 0,Y 549.052,Z 1149.49,A -85,B 0,C 180,E1 10358.729,E2 10358.729} C_VEL
LIN {X 0,Y 549.779,Z 1136.874,A -85,B 0,C 180,E1 10363.141,E2 10363.141} C_VEL
LIN {X 0,Y 551.159,Z 1119.491,A -85,B 0,C 180,E1 10367.394,E2 10367.394} C_VEL
LIN {X 0,Y 553.709,Z 1096.069,A -85,B 0,C 180,E1 10371.638,E2 10371.638} C_VEL
LIN {X 0,Y 557.573,Z 1065.919,A -85,B 0,C 180,E1 10375.77,E2 10375.77} C_VEL
LIN {X 0,Y 562.297,Z 1032.098,A -85,B 0,C 180,E1 10379.344,E2 10379.344} C_VEL
LIN {X 0,Y 567.2,Z 996.204,A -85,B 0,C 180,E1 10382.292,E2 10382.292} C_VEL
LIN {X 0,Y 572.339,Z 956.002,A -85,B 0,C 180,E1 10384.81,E2 10384.81} C_VEL
LIN {X 0,Y 576.995,Z 911.947,A -85,B 0,C 180,E1 10386.817,E2 10386.817} C_VEL
LIN {X 0,Y 580.696,Z 863.54,A -85,B 0,C 180,E1 10388.258,E2 10388.258} C_VEL
LIN {X 0,Y 580.624,Z 852.091,A -85,B 0,C 180,E1 10388.539,E2 10388.539} C_VEL
LIN {X 0,Y 562.618,Z 812.417,A -85,B 0,C 180,E1 10390.663,E2 10390.663} C_VEL
LIN {X 0,Y 547.737,Z 784.164,A -85,B 0,C 180,E1 10392.425,E2 10392.425} C_VEL
LIN {X 0,Y 547.7,Z 783.31,A -85,B 0,C 180,E1 10392.967,E2 10392.967} C_VEL
LIN {X 0,Y 547.56,Z 783.31,A -85,B 0,C 180,E1 10398.399,E2 10398.399} C_VEL
LIN {X 0,Y 547.573,Z 783.31,A -85,B 0,C 180,E1 10404.485,E2 10404.485} C_VEL
LIN {X 0,Y 547.771,Z 783.31,A -85,B 0,C 180,E1 10410.149,E2 10410.149} C_VEL
LIN {X 0,Y 548.006,Z 783.31,A -85,B 0,C 180,E1 10415.836,E2 10415.836} C_VEL
LIN {X 0,Y 548.048,Z 783.31,A -85,B 0,C 180,E1 10420.633,E2 10420.633} C_VEL
LIN {X 0,Y 548.12,Z 783.31,A -85,B 0,C 180,E1 10425.602,E2 10425.602} C_VEL
LIN {X 0,Y 548.302,Z 783.31,A -85,B 0,C 180,E1 10430.463,E2 10430.463} C_VEL
LIN {X 0,Y 548.524,Z 783.31,A -85,B 0,C 180,E1 10435.253,E2 10435.253} C_VEL
LIN {X 0,Y 548.598,Z 783.31,A -85,B 0,C 180,E1 10440.006,E2 10440.006} C_VEL
LIN {X 0,Y 548.513,Z 783.31,A -85,B 0,C 180,E1 10446.063,E2 10446.063} C_VEL
LIN {X 0,Y 548.306,Z 783.31,A -85,B 0,C 180,E1 10451.158,E2 10451.158} C_VEL
LIN {X 0,Y 548.15,Z 783.31,A -85,B 0,C 180,E1 10456.051,E2 10456.051} C_VEL
LIN {X 0,Y 547.966,Z 783.31,A -85,B 0,C 180,E1 10461.071,E2 10461.071} C_VEL
LIN {X 0,Y 547.819,Z 783.31,A -85,B 0,C 180,E1 10466.269,E2 10466.269} C_VEL
LIN {X 0,Y 547.731,Z 783.31,A -85,B 0,C 180,E1 10471.712,E2 10471.712} C_VEL
LIN {X 0,Y 547.584,Z 783.31,A -85,B 0,C 180,E1 10477.502,E2 10477.502} C_VEL
LIN {X 0,Y 547.566,Z 783.31,A -85,B 0,C 180,E1 10483.774,E2 10483.774} C_VEL
LIN {X 0,Y 547.553,Z 783.31,A -85,B 0,C 180,E1 10488.387,E2 10488.387} C_VEL
LIN {X 0,Y 547.554,Z 783.31,A -85,B 0,C 180,E1 10490.833,E2 10490.833} C_VEL
LIN {X 0,Y 551.781,Z 792.681,A -85,B 0,C 180,E1 10491.364,E2 10491.364} C_VEL
LIN {X 0,Y 578.536,Z 843.258,A -85,B 0,C 180,E1 10494.35,E2 10494.35} C_VEL
LIN {X 0,Y 580.911,Z 850.053,A -85,B 0,C 180,E1 10494.648,E2 10494.648} C_VEL
LIN {X 0,Y 578.271,Z 892.067,A -85,B 0,C 180,E1 10495.64,E2 10495.64} C_VEL
LIN {X 0,Y 574.588,Z 930.768,A -85,B 0,C 180,E1 10497.111,E2 10497.111} C_VEL
LIN {X 0,Y 569.908,Z 968.01,A -85,B 0,C 180,E1 10499.108,E2 10499.108} C_VEL
LIN {X 0,Y 564.508,Z 1005.132,A -85,B 0,C 180,E1 10501.834,E2 10501.834} C_VEL
LIN {X 0,Y 559.553,Z 1037.526,A -85,B 0,C 180,E1 10505.009,E2 10505.009} C_VEL
LIN {X 0,Y 555.022,Z 1067.312,A -85,B 0,C 180,E1 10508.888,E2 10508.888} C_VEL
LIN {X 0,Y 552.071,Z 1090.093,A -85,B 0,C 180,E1 10512.842,E2 10512.842} C_VEL
LIN {X 0,Y 550.051,Z 1108.704,A -85,B 0,C 180,E1 10517.271,E2 10517.271} C_VEL
LIN {X 0,Y 549.217,Z 1120.251,A -85,B 0,C 180,E1 10521.274,E2 10521.274} C_VEL
LIN {X 0,Y 548.878,Z 1127.438,A -85,B 0,C 180,E1 10525.251,E2 10525.251} C_VEL
LIN {X 0,Y 548.929,Z 1130.374,A -85,B 0,C 180,E1 10530.001,E2 10530.001} C_VEL
LIN {X 0,Y 548.898,Z 1127.328,A -85,B 0,C 180,E1 10534.752,E2 10534.752} C_VEL
LIN {X 0,Y 549.234,Z 1120.041,A -85,B 0,C 180,E1 10538.728,E2 10538.728} C_VEL
LIN {X 0,Y 550.146,Z 1106.878,A -85,B 0,C 180,E1 10543.134,E2 10543.134} C_VEL
LIN {X 0,Y 552.104,Z 1088.574,A -85,B 0,C 180,E1 10547.366,E2 10547.366} C_VEL
LIN {X 0,Y 555.373,Z 1064.396,A -85,B 0,C 180,E1 10551.455,E2 10551.455} C_VEL
LIN {X 0,Y 559.735,Z 1036.321,A -85,B 0,C 180,E1 10555.034,E2 10555.034} C_VEL
LIN {X 0,Y 565.028,Z 1002.09,A -85,B 0,C 180,E1 10558.329,E2 10558.329} C_VEL
LIN {X 0,Y 570.372,Z 965.147,A -85,B 0,C 180,E1 10560.978,E2 10560.978} C_VEL
LIN {X 0,Y 575.141,Z 925.757,A -85,B 0,C 180,E1 10563.026,E2 10563.026} C_VEL
LIN {X 0,Y 578.886,Z 883.002,A -85,B 0,C 180,E1 10564.54,E2 10564.54} C_VEL
LIN {X 0,Y 580.407,Z 847.165,A -85,B 0,C 180,E1 10565.346,E2 10565.346} C_VEL
LIN {X 0,Y 554.505,Z 797.281,A -85,B 0,C 180,E1 10568.227,E2 10568.227} C_VEL
LIN {X 0,Y 547.653,Z 783.84,A -85,B 0,C 180,E1 10569.049,E2 10569.049} C_VEL
LIN {X 0,Y 547.558,Z 783.31,A -85,B 0,C 180,E1 10573.988,E2 10573.988} C_VEL
LIN {X 0,Y 547.556,Z 783.31,A -85,B 0,C 180,E1 10580.47,E2 10580.47} C_VEL
LIN {X 0,Y 547.588,Z 783.31,A -85,B 0,C 180,E1 10586.396,E2 10586.396} C_VEL
LIN {X 0,Y 547.856,Z 783.31,A -85,B 0,C 180,E1 10592.254,E2 10592.254} C_VEL
LIN {X 0,Y 547.948,Z 783.31,A -85,B 0,C 180,E1 10597.22,E2 10597.22} C_VEL
LIN {X 0,Y 548.118,Z 783.31,A -85,B 0,C 180,E1 10602.293,E2 10602.293} C_VEL
LIN {X 0,Y 548.214,Z 783.31,A -85,B 0,C 180,E1 10607.221,E2 10607.221} C_VEL
LIN {X 0,Y 548.47,Z 783.31,A -85,B 0,C 180,E1 10612.188,E2 10612.188} C_VEL
LIN {X 0,Y 548.597,Z 783.31,A -85,B 0,C 180,E1 10616.828,E2 10616.828} C_VEL
LIN {X 0,Y 548.718,Z 783.31,A -85,B 0,C 180,E1 10621.576,E2 10621.576} C_VEL
LIN {X 0,Y 548.491,Z 783.31,A -85,B 0,C 180,E1 10626.337,E2 10626.337} C_VEL
LIN {X 0,Y 548.327,Z 783.31,A -85,B 0,C 180,E1 10631.146,E2 10631.146} C_VEL
LIN {X 0,Y 548.176,Z 783.31,A -85,B 0,C 180,E1 10636.038,E2 10636.038} C_VEL
LIN {X 0,Y 547.998,Z 783.31,A -85,B 0,C 180,E1 10641.057,E2 10641.057} C_VEL
LIN {X 0,Y 547.883,Z 783.31,A -85,B 0,C 180,E1 10646.253,E2 10646.253} C_VEL
LIN {X 0,Y 547.789,Z 783.31,A -85,B 0,C 180,E1 10651.694,E2 10651.694} C_VEL
LIN {X 0,Y 547.566,Z 783.31,A -85,B 0,C 180,E1 10657.488,E2 10657.488} C_VEL
LIN {X 0,Y 547.462,Z 783.31,A -85,B 0,C 180,E1 10663.768,E2 10663.768} C_VEL
LIN {X 0,Y 547.563,Z 783.757,A -85,B 0,C 180,E1 10667.56,E2 10667.56} C_VEL
LIN {X 0,Y 574.697,Z 837.495,A -85,B 0,C 180,E1 10670.724,E2 10670.724} C_VEL
LIN {X 0,Y 581.311,Z 854.492,A -85,B 0,C 180,E1 10671.572,E2 10671.572} C_VEL
LIN {X 0,Y 578.12,Z 898.316,A -85,B 0,C 180,E1 10672.702,E2 10672.702} C_VEL
LIN {X 0,Y 573.708,Z 943.407,A -85,B 0,C 180,E1 10674.535,E2 10674.535} C_VEL
LIN {X 0,Y 568.457,Z 986.626,A -85,B 0,C 180,E1 10677.033,E2 10677.033} C_VEL
LIN {X 0,Y 565.886,Z 1006.093,A -85,B 0,C 180,E1 10678.449,E2 10678.449} C_VEL
LIN {X 0,Y 560.327,Z 1020.025,A -85,B 0,C 180,E1 10679.385,E2 10679.385} C_VEL
LIN {X 0,Y 554.878,Z 1033.351,A -85,B 0,C 180,E1 10680.402,E2 10680.402} C_VEL
LIN {X 0,Y 550.158,Z 1065.474,A -85,B 0,C 180,E1 10683.853,E2 10683.853} C_VEL
LIN {X 0,Y 546.239,Z 1094.857,A -85,B 0,C 180,E1 10687.924,E2 10687.924} C_VEL
LIN {X 0,Y 543.405,Z 1119.124,A -85,B 0,C 180,E1 10692.347,E2 10692.347} C_VEL
LIN {X 0,Y 541.913,Z 1136.583,A -85,B 0,C 180,E1 10696.662,E2 10696.662} C_VEL
LIN {X 0,Y 541.213,Z 1149.237,A -85,B 0,C 180,E1 10701.141,E2 10701.141} C_VEL
LIN {X 0,Y 540.977,Z 1156.025,A -85,B 0,C 180,E1 10705.179,E2 10705.179} C_VEL
LIN {X 0,Y 540.957,Z 1158.958,A -85,B 0,C 180,E1 10709.999,E2 10709.999} C_VEL
LIN {X 0,Y 540.987,Z 1156.023,A -85,B 0,C 180,E1 10714.818,E2 10714.818} C_VEL
LIN {X 0,Y 541.173,Z 1149.242,A -85,B 0,C 180,E1 10718.857,E2 10718.857} C_VEL
LIN {X 0,Y 541.943,Z 1136.577,A -85,B 0,C 180,E1 10723.334,E2 10723.334} C_VEL
LIN {X 0,Y 543.437,Z 1119.124,A -85,B 0,C 180,E1 10727.649,E2 10727.649} C_VEL
LIN {X 0,Y 546.233,Z 1094.855,A -85,B 0,C 180,E1 10732.076,E2 10732.076} C_VEL
LIN {X 0,Y 550.399,Z 1064.125,A -85,B 0,C 180,E1 10736.314,E2 10736.314} C_VEL
LIN {X 0,Y 555.691,Z 1028.436,A -85,B 0,C 180,E1 10740.066,E2 10740.066} C_VEL
LIN {X 0,Y 561.411,Z 988.081,A -85,B 0,C 180,E1 10743.286,E2 10743.286} C_VEL
LIN {X 0,Y 566.608,Z 947.624,A -85,B 0,C 180,E1 10745.687,E2 10745.687} C_VEL
LIN {X 0,Y 571.003,Z 906.438,A -85,B 0,C 180,E1 10747.467,E2 10747.467} C_VEL
LIN {X 0,Y 574.403,Z 861.753,A -85,B 0,C 180,E1 10748.765,E2 10748.765} C_VEL
LIN {X 0,Y 574.176,Z 854.528,A -85,B 0,C 180,E1 10748.959,E2 10748.959} C_VEL
LIN {X 0,Y 556.842,Z 816.225,A -85,B 0,C 180,E1 10751.079,E2 10751.079} C_VEL
LIN {X 0,Y 539.836,Z 784.193,A -85,B 0,C 180,E1 10753.149,E2 10753.149} C_VEL
LIN {X 0,Y 539.746,Z 783.31,A -85,B 0,C 180,E1 10753.457,E2 10753.457} C_VEL
LIN {X 0,Y 539.602,Z 783.31,A -85,B 0,C 180,E1 10759.785,E2 10759.785} C_VEL
LIN {X 0,Y 539.699,Z 783.31,A -85,B 0,C 180,E1 10765.852,E2 10765.852} C_VEL
LIN {X 0,Y 539.88,Z 783.31,A -85,B 0,C 180,E1 10771.513,E2 10771.513} C_VEL
LIN {X 0,Y 540.068,Z 783.31,A -85,B 0,C 180,E1 10776.882,E2 10776.882} C_VEL
LIN {X 0,Y 540.212,Z 783.31,A -85,B 0,C 180,E1 10782.476,E2 10782.476} C_VEL
LIN {X 0,Y 540.348,Z 783.31,A -85,B 0,C 180,E1 10788.93,E2 10788.93} C_VEL
LIN {X 0,Y 540.55,Z 783.31,A -85,B 0,C 180,E1 10793.569,E2 10793.569} C_VEL
LIN {X 0,Y 540.681,Z 783.31,A -85,B 0,C 180,E1 10798.4,E2 10798.4} C_VEL
LIN {X 0,Y 540.644,Z 783.31,A -85,B 0,C 180,E1 10803.219,E2 10803.219} C_VEL
LIN {X 0,Y 540.483,Z 783.31,A -85,B 0,C 180,E1 10808.063,E2 10808.063} C_VEL
LIN {X 0,Y 540.322,Z 783.31,A -85,B 0,C 180,E1 10812.969,E2 10812.969} C_VEL
LIN {X 0,Y 540.181,Z 783.31,A -85,B 0,C 180,E1 10817.976,E2 10817.976} C_VEL
LIN {X 0,Y 540.007,Z 783.31,A -85,B 0,C 180,E1 10823.134,E2 10823.134} C_VEL
LIN {X 0,Y 539.828,Z 783.31,A -85,B 0,C 180,E1 10828.503,E2 10828.503} C_VEL
LIN {X 0,Y 539.706,Z 783.31,A -85,B 0,C 180,E1 10834.162,E2 10834.162} C_VEL
LIN {X 0,Y 539.613,Z 783.31,A -85,B 0,C 180,E1 10840.23,E2 10840.23} C_VEL
LIN {X 0,Y 539.586,Z 783.31,A -85,B 0,C 180,E1 10845.414,E2 10845.414} C_VEL
LIN {X 0,Y 539.604,Z 783.364,A -85,B 0,C 180,E1 10850.1,E2 10850.1} C_VEL
LIN {X 0,Y 542.191,Z 789.089,A -85,B 0,C 180,E1 10850.437,E2 10850.437} C_VEL
LIN {X 0,Y 571.075,Z 843.701,A -85,B 0,C 180,E1 10853.781,E2 10853.781} C_VEL
LIN {X 0,Y 574.546,Z 851.96,A -85,B 0,C 180,E1 10854.203,E2 10854.203} C_VEL
LIN {X 0,Y 571.681,Z 895.215,A -85,B 0,C 180,E1 10855.266,E2 10855.266} C_VEL
LIN {X 0,Y 567.233,Z 937.638,A -85,B 0,C 180,E1 10856.966,E2 10856.966} C_VEL
LIN {X 0,Y 561.795,Z 977.892,A -85,B 0,C 180,E1 10859.311,E2 10859.311} C_VEL
LIN {X 0,Y 556.162,Z 1014.142,A -85,B 0,C 180,E1 10862.215,E2 10862.215} C_VEL
LIN {X 0,Y 550.656,Z 1047.823,A -85,B 0,C 180,E1 10865.841,E2 10865.841} C_VEL
LIN {X 0,Y 546.521,Z 1074.825,A -85,B 0,C 180,E1 10869.725,E2 10869.725} C_VEL
LIN {X 0,Y 543.521,Z 1097.288,A -85,B 0,C 180,E1 10874.074,E2 10874.074} C_VEL
LIN {X 0,Y 541.799,Z 1114.22,A -85,B 0,C 180,E1 10878.712,E2 10878.712} C_VEL
LIN {X 0,Y 541.141,Z 1123.865,A -85,B 0,C 180,E1 10882.763,E2 10882.763} C_VEL
LIN {X 0,Y 540.98,Z 1129.296,A -85,B 0,C 180,E1 10886.79,E2 10886.79} C_VEL
LIN {X 0,Y 541.04,Z 1130.581,A -85,B 0,C 180,E1 10890.001,E2 10890.001} C_VEL
LIN {X 0,Y 541.018,Z 1127.553,A -85,B 0,C 180,E1 10894.821,E2 10894.821} C_VEL
LIN {X 0,Y 541.378,Z 1120.302,A -85,B 0,C 180,E1 10898.856,E2 10898.856} C_VEL
LIN {X 0,Y 542.263,Z 1108.679,A -85,B 0,C 180,E1 10902.918,E2 10902.918} C_VEL
LIN {X 0,Y 544.316,Z 1089.958,A -85,B 0,C 180,E1 10907.413,E2 10907.413} C_VEL
LIN {X 0,Y 547.824,Z 1065.349,A -85,B 0,C 180,E1 10911.676,E2 10911.676} C_VEL
LIN {X 0,Y 552.558,Z 1036.152,A -85,B 0,C 180,E1 10915.447,E2 10915.447} C_VEL
LIN {X 0,Y 557.996,Z 1002.689,A -85,B 0,C 180,E1 10918.705,E2 10918.705} C_VEL
LIN {X 0,Y 563.584,Z 965.668,A -85,B 0,C 180,E1 10921.393,E2 10921.393} C_VEL
LIN {X 0,Y 568.561,Z 926.4,A -85,B 0,C 180,E1 10923.458,E2 10923.458} C_VEL
LIN {X 0,Y 572.425,Z 884.337,A -85,B 0,C 180,E1 10924.972,E2 10924.972} C_VEL
LIN {X 0,Y 574.219,Z 850.122,A -85,B 0,C 180,E1 10925.765,E2 10925.765} C_VEL
LIN {X 0,Y 547.876,Z 799.282,A -85,B 0,C 180,E1 10928.779,E2 10928.779} C_VEL
LIN {X 0,Y 539.845,Z 784.77,A -85,B 0,C 180,E1 10929.754,E2 10929.754} C_VEL
LIN {X 0,Y 539.673,Z 783.31,A -85,B 0,C 180,E1 10929.844,E2 10929.844} C_VEL
LIN {X 0,Y 539.591,Z 783.31,A -85,B 0,C 180,E1 10935.409,E2 10935.409} C_VEL
LIN {X 0,Y 539.61,Z 783.31,A -85,B 0,C 180,E1 10941.846,E2 10941.846} C_VEL
LIN {X 0,Y 539.734,Z 783.31,A -85,B 0,C 180,E1 10947.762,E2 10947.762} C_VEL
LIN {X 0,Y 539.961,Z 783.31,A -85,B 0,C 180,E1 10953.892,E2 10953.892} C_VEL
LIN {X 0,Y 540.051,Z 783.31,A -85,B 0,C 180,E1 10958.605,E2 10958.605} C_VEL
LIN {X 0,Y 540.182,Z 783.31,A -85,B 0,C 180,E1 10963.706,E2 10963.706} C_VEL
LIN {X 0,Y 540.396,Z 783.31,A -85,B 0,C 180,E1 10968.918,E2 10968.918} C_VEL
LIN {X 0,Y 540.591,Z 783.31,A -85,B 0,C 180,E1 10973.557,E2 10973.557} C_VEL
LIN {X 0,Y 540.706,Z 783.31,A -85,B 0,C 180,E1 10978.388,E2 10978.388} C_VEL
LIN {X 0,Y 540.656,Z 783.31,A -85,B 0,C 180,E1 10983.207,E2 10983.207} C_VEL
LIN {X 0,Y 540.496,Z 783.31,A -85,B 0,C 180,E1 10988.051,E2 10988.051} C_VEL
LIN {X 0,Y 540.332,Z 783.31,A -85,B 0,C 180,E1 10992.956,E2 10992.956} C_VEL
LIN {X 0,Y 540.229,Z 783.31,A -85,B 0,C 180,E1 10997.962,E2 10997.962} C_VEL
LIN {X 0,Y 540.025,Z 783.31,A -85,B 0,C 180,E1 11003.12,E2 11003.12} C_VEL
LIN {X 0,Y 539.887,Z 783.31,A -85,B 0,C 180,E1 11008.486,E2 11008.486} C_VEL
LIN {X 0,Y 539.724,Z 783.31,A -85,B 0,C 180,E1 11014.146,E2 11014.146} C_VEL
LIN {X 0,Y 539.565,Z 783.31,A -85,B 0,C 180,E1 11020.218,E2 11020.218} C_VEL
LIN {X 0,Y 539.617,Z 783.31,A -85,B 0,C 180,E1 11026.779,E2 11026.779} C_VEL
LIN {X 0,Y 547.031,Z 798.24,A -85,B 0,C 180,E1 11027.767,E2 11027.767} C_VEL
LIN {X 0,Y 568.173,Z 839.77,A -85,B 0,C 180,E1 11030.264,E2 11030.264} C_VEL
LIN {X 0,Y 574.809,Z 857.881,A -85,B 0,C 180,E1 11031.174,E2 11031.174} C_VEL
LIN {X 0,Y 571.499,Z 900.201,A -85,B 0,C 180,E1 11032.31,E2 11032.31} C_VEL
LIN {X 0,Y 567.001,Z 943.804,A -85,B 0,C 180,E1 11034.111,E2 11034.111} C_VEL
LIN {X 0,Y 561.549,Z 986.897,A -85,B 0,C 180,E1 11036.634,E2 11036.634} C_VEL
LIN {X 0,Y 555.814,Z 1027.252,A -85,B 0,C 180,E1 11039.826,E2 11039.826} C_VEL
LIN {X 0,Y 554.878,Z 1033.351,A -85,B 0,C 180,E1 11040.402,E2 11040.402} C_VEL
LIN {X 0,Y 549.326,Z 1046.214,A -85,B 0,C 180,E1 11041.505,E2 11041.505} C_VEL
LIN {X 0,Y 544.178,Z 1056.988,A -85,B 0,C 180,E1 11042.519,E2 11042.519} C_VEL
LIN {X 0,Y 543.896,Z 1058.435,A -85,B 0,C 180,E1 11042.687,E2 11042.687} C_VEL
LIN {X 0,Y 539.643,Z 1087.45,A -85,B 0,C 180,E1 11046.518,E2 11046.518} C_VEL
LIN {X 0,Y 536.307,Z 1113.262,A -85,B 0,C 180,E1 11050.945,E2 11050.945} C_VEL
LIN {X 0,Y 534.267,Z 1133.432,A -85,B 0,C 180,E1 11055.631,E2 11055.631} C_VEL
LIN {X 0,Y 533.405,Z 1147.017,A -85,B 0,C 180,E1 11060.186,E2 11060.186} C_VEL
LIN {X 0,Y 533.172,Z 1154.271,A -85,B 0,C 180,E1 11063.948,E2 11063.948} C_VEL
LIN {X 0,Y 532.998,Z 1158.405,A -85,B 0,C 180,E1 11068.37,E2 11068.37} C_VEL
LIN {X 0,Y 532.984,Z 1158.405,A -85,B 0,C 180,E1 11071.628,E2 11071.628} C_VEL
LIN {X 0,Y 533.153,Z 1153.537,A -85,B 0,C 180,E1 11076.526,E2 11076.526} C_VEL
LIN {X 0,Y 533.574,Z 1143.889,A -85,B 0,C 180,E1 11081.049,E2 11081.049} C_VEL
LIN {X 0,Y 534.763,Z 1128.721,A -85,B 0,C 180,E1 11085.605,E2 11085.605} C_VEL
LIN {X 0,Y 537.077,Z 1107.107,A -85,B 0,C 180,E1 11090.216,E2 11090.216} C_VEL
LIN {X 0,Y 540.569,Z 1080.784,A -85,B 0,C 180,E1 11094.448,E2 11094.448} C_VEL
LIN {X 0,Y 545.146,Z 1049.528,A -85,B 0,C 180,E1 11098.33,E2 11098.33} C_VEL
LIN {X 0,Y 550.731,Z 1013.841,A -85,B 0,C 180,E1 11101.745,E2 11101.745} C_VEL
LIN {X 0,Y 556.613,Z 973.263,A -85,B 0,C 180,E1 11104.694,E2 11104.694} C_VEL
LIN {X 0,Y 562.252,Z 928.05,A -85,B 0,C 180,E1 11107.084,E2 11107.084} C_VEL
LIN {X 0,Y 566.902,Z 880.504,A -85,B 0,C 180,E1 11108.771,E2 11108.771} C_VEL
LIN {X 0,Y 567.737,Z 856.906,A -85,B 0,C 180,E1 11109.393,E2 11109.393} C_VEL
LIN {X 0,Y 550.786,Z 819.376,A -85,B 0,C 180,E1 11111.542,E2 11111.542} C_VEL
LIN {X 0,Y 531.929,Z 784.67,A -85,B 0,C 180,E1 11113.896,E2 11113.896} C_VEL
LIN {X 0,Y 531.821,Z 783.31,A -85,B 0,C 180,E1 11113.939,E2 11113.939} C_VEL
LIN {X 0,Y 531.648,Z 783.31,A -85,B 0,C 180,E1 11120.305,E2 11120.305} C_VEL
LIN {X 0,Y 531.806,Z 783.31,A -85,B 0,C 180,E1 11125.711,E2 11125.711} C_VEL
LIN {X 0,Y 531.953,Z 783.31,A -85,B 0,C 180,E1 11132,E2 11132} C_VEL
LIN {X 0,Y 532.115,Z 783.31,A -85,B 0,C 180,E1 11136.516,E2 11136.516} C_VEL
LIN {X 0,Y 532.244,Z 783.31,A -85,B 0,C 180,E1 11141.76,E2 11141.76} C_VEL
LIN {X 0,Y 532.32,Z 783.31,A -85,B 0,C 180,E1 11146.845,E2 11146.845} C_VEL
LIN {X 0,Y 532.598,Z 783.31,A -85,B 0,C 180,E1 11151.829,E2 11151.829} C_VEL
LIN {X 0,Y 532.771,Z 783.31,A -85,B 0,C 180,E1 11156.746,E2 11156.746} C_VEL
LIN {X 0,Y 532.886,Z 783.31,A -85,B 0,C 180,E1 11161.635,E2 11161.635} C_VEL
LIN {X 0,Y 532.652,Z 783.31,A -85,B 0,C 180,E1 11166.539,E2 11166.539} C_VEL
LIN {X 0,Y 532.455,Z 783.31,A -85,B 0,C 180,E1 11171.495,E2 11171.495} C_VEL
LIN {X 0,Y 532.312,Z 783.31,A -85,B 0,C 180,E1 11176.542,E2 11176.542} C_VEL
LIN {X 0,Y 532.114,Z 783.31,A -85,B 0,C 180,E1 11181.73,E2 11181.73} C_VEL
LIN {X 0,Y 531.893,Z 783.31,A -85,B 0,C 180,E1 11187.988,E2 11187.988} C_VEL
LIN {X 0,Y 531.793,Z 783.31,A -85,B 0,C 180,E1 11194.287,E2 11194.287} C_VEL
LIN {X 0,Y 531.654,Z 783.31,A -85,B 0,C 180,E1 11199.696,E2 11199.696} C_VEL
LIN {X 0,Y 531.683,Z 783.31,A -85,B 0,C 180,E1 11205.437,E2 11205.437} C_VEL
LIN {X 0,Y 531.718,Z 783.959,A -85,B 0,C 180,E1 11209.35,E2 11209.35} C_VEL
LIN {X 0,Y 562.66,Z 842.109,A -85,B 0,C 180,E1 11213.079,E2 11213.079} C_VEL
LIN {X 0,Y 568.104,Z 853.442,A -85,B 0,C 180,E1 11213.736,E2 11213.736} C_VEL
LIN {X 0,Y 565.208,Z 896.499,A -85,B 0,C 180,E1 11214.827,E2 11214.827} C_VEL
LIN {X 0,Y 560.591,Z 938.661,A -85,B 0,C 180,E1 11216.547,E2 11216.547} C_VEL
LIN {X 0,Y 555.015,Z 978.195,A -85,B 0,C 180,E1 11218.883,E2 11218.883} C_VEL
LIN {X 0,Y 548.966,Z 1015.398,A -85,B 0,C 180,E1 11221.907,E2 11221.907} C_VEL
LIN {X 0,Y 543.32,Z 1048.155,A -85,B 0,C 180,E1 11225.494,E2 11225.494} C_VEL
LIN {X 0,Y 539.005,Z 1075.135,A -85,B 0,C 180,E1 11229.43,E2 11229.43} C_VEL
LIN {X 0,Y 535.764,Z 1097.93,A -85,B 0,C 180,E1 11233.925,E2 11233.925} C_VEL
LIN {X 0,Y 533.962,Z 1114.485,A -85,B 0,C 180,E1 11238.545,E2 11238.545} C_VEL
LIN {X 0,Y 533.261,Z 1124.107,A -85,B 0,C 180,E1 11242.656,E2 11242.656} C_VEL
LIN {X 0,Y 533.08,Z 1129.509,A -85,B 0,C 180,E1 11246.743,E2 11246.743} C_VEL
LIN {X 0,Y 533.141,Z 1130.789,A -85,B 0,C 180,E1 11250.001,E2 11250.001} C_VEL
LIN {X 0,Y 533.127,Z 1127.778,A -85,B 0,C 180,E1 11254.892,E2 11254.892} C_VEL
LIN {X 0,Y 533.515,Z 1120.556,A -85,B 0,C 180,E1 11258.988,E2 11258.988} C_VEL
LIN {X 0,Y 534.46,Z 1108.959,A -85,B 0,C 180,E1 11263.11,E2 11263.11} C_VEL
LIN {X 0,Y 536.676,Z 1090.26,A -85,B 0,C 180,E1 11267.669,E2 11267.669} C_VEL
LIN {X 0,Y 540.252,Z 1066.311,A -85,B 0,C 180,E1 11271.899,E2 11271.899} C_VEL
LIN {X 0,Y 545.296,Z 1036.748,A -85,B 0,C 180,E1 11275.784,E2 11275.784} C_VEL
LIN {X 0,Y 551.032,Z 1003.112,A -85,B 0,C 180,E1 11279.102,E2 11279.102} C_VEL
LIN {X 0,Y 557.077,Z 964.529,A -85,B 0,C 180,E1 11281.917,E2 11281.917} C_VEL
LIN {X 0,Y 562.235,Z 924.904,A -85,B 0,C 180,E1 11284.001,E2 11284.001} C_VEL
LIN {X 0,Y 566.295,Z 882.309,A -85,B 0,C 180,E1 11285.512,E2 11285.512} C_VEL
LIN {X 0,Y 567.79,Z 852.75,A -85,B 0,C 180,E1 11286.21,E2 11286.21} C_VEL
LIN {X 0,Y 542.845,Z 804.267,A -85,B 0,C 180,E1 11289.154,E2 11289.154} C_VEL
LIN {X 0,Y 531.813,Z 784.294,A -85,B 0,C 180,E1 11290.534,E2 11290.534} C_VEL
LIN {X 0,Y 531.76,Z 783.31,A -85,B 0,C 180,E1 11290.69,E2 11290.69} C_VEL
LIN {X 0,Y 531.683,Z 783.31,A -85,B 0,C 180,E1 11296.844,E2 11296.844} C_VEL
LIN {X 0,Y 531.635,Z 783.31,A -85,B 0,C 180,E1 11303.234,E2 11303.234} C_VEL
LIN {X 0,Y 531.852,Z 783.31,A -85,B 0,C 180,E1 11309.146,E2 11309.146} C_VEL
LIN {X 0,Y 532.028,Z 783.31,A -85,B 0,C 180,E1 11314.707,E2 11314.707} C_VEL
LIN {X 0,Y 532.208,Z 783.31,A -85,B 0,C 180,E1 11320.019,E2 11320.019} C_VEL
LIN {X 0,Y 532.355,Z 783.31,A -85,B 0,C 180,E1 11325.401,E2 11325.401} C_VEL
LIN {X 0,Y 532.653,Z 783.31,A -85,B 0,C 180,E1 11331.818,E2 11331.818} C_VEL
LIN {X 0,Y 532.781,Z 783.31,A -85,B 0,C 180,E1 11336.734,E2 11336.734} C_VEL
LIN {X 0,Y 532.908,Z 783.31,A -85,B 0,C 180,E1 11341.623,E2 11341.623} C_VEL
LIN {X 0,Y 532.658,Z 783.31,A -85,B 0,C 180,E1 11346.527,E2 11346.527} C_VEL
LIN {X 0,Y 532.485,Z 783.31,A -85,B 0,C 180,E1 11351.482,E2 11351.482} C_VEL
LIN {X 0,Y 532.352,Z 783.31,A -85,B 0,C 180,E1 11356.528,E2 11356.528} C_VEL
LIN {X 0,Y 532.148,Z 783.31,A -85,B 0,C 180,E1 11361.716,E2 11361.716} C_VEL
LIN {X 0,Y 531.952,Z 783.31,A -85,B 0,C 180,E1 11367.994,E2 11367.994} C_VEL
LIN {X 0,Y 531.828,Z 783.31,A -85,B 0,C 180,E1 11374.287,E2 11374.287} C_VEL
LIN {X 0,Y 531.638,Z 783.31,A -85,B 0,C 180,E1 11380.945,E2 11380.945} C_VEL
LIN {X 0,Y 531.682,Z 783.31,A -85,B 0,C 180,E1 11386.051,E2 11386.051} C_VEL
LIN {X 0,Y 534.345,Z 789.196,A -85,B 0,C 180,E1 11386.431,E2 11386.431} C_VEL
LIN {X 0,Y 559.91,Z 837.935,A -85,B 0,C 180,E1 11389.567,E2 11389.567} C_VEL
LIN {X 0,Y 568.365,Z 860.078,A -85,B 0,C 180,E1 11390.739,E2 11390.739} C_VEL
LIN {X 0,Y 564.753,Z 903.705,A -85,B 0,C 180,E1 11391.966,E2 11391.966} C_VEL
LIN {X 0,Y 560.217,Z 945.194,A -85,B 0,C 180,E1 11393.73,E2 11393.73} C_VEL
LIN {X 0,Y 554.559,Z 987.787,A -85,B 0,C 180,E1 11396.266,E2 11396.266} C_VEL
LIN {X 0,Y 548.634,Z 1027.668,A -85,B 0,C 180,E1 11399.473,E2 11399.473} C_VEL
LIN {X 0,Y 543.896,Z 1058.435,A -85,B 0,C 180,E1 11402.687,E2 11402.687} C_VEL
LIN {X 0,Y 540.239,Z 1067.289,A -85,B 0,C 180,E1 11403.646,E2 11403.646} C_VEL
LIN {X 0,Y 533.25,Z 1079.811,A -85,B 0,C 180,E1 11405.101,E2 11405.101} C_VEL
LIN {X 0,Y 532.979,Z 1081.122,A -85,B 0,C 180,E1 11405.285,E2 11405.285} C_VEL
LIN {X 0,Y 529.446,Z 1106.763,A -85,B 0,C 180,E1 11409.476,E2 11409.476} C_VEL
LIN {X 0,Y 526.921,Z 1128.429,A -85,B 0,C 180,E1 11414.164,E2 11414.164} C_VEL
LIN {X 0,Y 525.758,Z 1143.662,A -85,B 0,C 180,E1 11418.798,E2 11418.798} C_VEL
LIN {X 0,Y 525.285,Z 1153.314,A -85,B 0,C 180,E1 11423.373,E2 11423.373} C_VEL
LIN {X 0,Y 525.122,Z 1158.198,A -85,B 0,C 180,E1 11428.345,E2 11428.345} C_VEL
LIN {X 0,Y 525.11,Z 1158.198,A -85,B 0,C 180,E1 11431.652,E2 11431.652} C_VEL
LIN {X 0,Y 525.244,Z 1153.311,A -85,B 0,C 180,E1 11436.625,E2 11436.625} C_VEL
LIN {X 0,Y 525.703,Z 1143.745,A -85,B 0,C 180,E1 11441.172,E2 11441.172} C_VEL
LIN {X 0,Y 526.962,Z 1128.401,A -85,B 0,C 180,E1 11445.842,E2 11445.842} C_VEL
LIN {X 0,Y 529.455,Z 1106.775,A -85,B 0,C 180,E1 11450.52,E2 11450.52} C_VEL
LIN {X 0,Y 533.094,Z 1080.545,A -85,B 0,C 180,E1 11454.797,E2 11454.797} C_VEL
LIN {X 0,Y 537.776,Z 1050.322,A -85,B 0,C 180,E1 11458.616,E2 11458.616} C_VEL
LIN {X 0,Y 543.781,Z 1013.407,A -85,B 0,C 180,E1 11462.199,E2 11462.199} C_VEL
LIN {X 0,Y 549.962,Z 972.193,A -85,B 0,C 180,E1 11465.214,E2 11465.214} C_VEL
LIN {X 0,Y 555.772,Z 928.038,A -85,B 0,C 180,E1 11467.557,E2 11467.557} C_VEL
LIN {X 0,Y 560.57,Z 880.533,A -85,B 0,C 180,E1 11469.258,E2 11469.258} C_VEL
LIN {X 0,Y 561.284,Z 859.231,A -85,B 0,C 180,E1 11469.842,E2 11469.842} C_VEL
LIN {X 0,Y 545.024,Z 822.982,A -85,B 0,C 180,E1 11471.984,E2 11471.984} C_VEL
LIN {X 0,Y 523.866,Z 784.021,A -85,B 0,C 180,E1 11474.712,E2 11474.712} C_VEL
LIN {X 0,Y 523.746,Z 783.31,A -85,B 0,C 180,E1 11480.485,E2 11480.485} C_VEL
LIN {X 0,Y 523.923,Z 783.31,A -85,B 0,C 180,E1 11486.997,E2 11486.997} C_VEL
LIN {X 0,Y 524.075,Z 783.31,A -85,B 0,C 180,E1 11492.456,E2 11492.456} C_VEL
LIN {X 0,Y 524.215,Z 783.31,A -85,B 0,C 180,E1 11497.938,E2 11497.938} C_VEL
LIN {X 0,Y 524.358,Z 783.31,A -85,B 0,C 180,E1 11503.213,E2 11503.213} C_VEL
LIN {X 0,Y 524.494,Z 783.31,A -85,B 0,C 180,E1 11509.164,E2 11509.164} C_VEL
LIN {X 0,Y 524.812,Z 783.31,A -85,B 0,C 180,E1 11515.038,E2 11515.038} C_VEL
LIN {X 0,Y 524.955,Z 783.31,A -85,B 0,C 180,E1 11520.006,E2 11520.006} C_VEL
LIN {X 0,Y 524.868,Z 783.31,A -85,B 0,C 180,E1 11524.974,E2 11524.974} C_VEL
LIN {X 0,Y 524.532,Z 783.31,A -85,B 0,C 180,E1 11530.858,E2 11530.858} C_VEL
LIN {X 0,Y 524.371,Z 783.31,A -85,B 0,C 180,E1 11536.8,E2 11536.8} C_VEL
LIN {X 0,Y 524.146,Z 783.31,A -85,B 0,C 180,E1 11542.331,E2 11542.331} C_VEL
LIN {X 0,Y 524.016,Z 783.31,A -85,B 0,C 180,E1 11547.561,E2 11547.561} C_VEL
LIN {X 0,Y 523.879,Z 783.31,A -85,B 0,C 180,E1 11553.338,E2 11553.338} C_VEL
LIN {X 0,Y 523.751,Z 783.31,A -85,B 0,C 180,E1 11559.53,E2 11559.53} C_VEL
LIN {X 0,Y 523.757,Z 783.31,A -85,B 0,C 180,E1 11566.031,E2 11566.031} C_VEL
LIN {X 0,Y 523.751,Z 783.31,A -85,B 0,C 180,E1 11568.506,E2 11568.506} C_VEL
LIN {X 0,Y 526.439,Z 789.248,A -85,B 0,C 180,E1 11568.916,E2 11568.916} C_VEL
LIN {X 0,Y 553.97,Z 839.827,A -85,B 0,C 180,E1 11572.312,E2 11572.312} C_VEL
LIN {X 0,Y 561.708,Z 857.669,A -85,B 0,C 180,E1 11573.327,E2 11573.327} C_VEL
LIN {X 0,Y 558.63,Z 899.283,A -85,B 0,C 180,E1 11574.437,E2 11574.437} C_VEL
LIN {X 0,Y 553.929,Z 939.859,A -85,B 0,C 180,E1 11576.131,E2 11576.131} C_VEL
LIN {X 0,Y 548.114,Z 979.262,A -85,B 0,C 180,E1 11578.497,E2 11578.497} C_VEL
LIN {X 0,Y 541.9,Z 1015.762,A -85,B 0,C 180,E1 11581.507,E2 11581.507} C_VEL
LIN {X 0,Y 536.019,Z 1048.474,A -85,B 0,C 180,E1 11585.137,E2 11585.137} C_VEL
LIN {X 0,Y 531.502,Z 1075.428,A -85,B 0,C 180,E1 11589.126,E2 11589.126} C_VEL
LIN {X 0,Y 528.073,Z 1098.194,A -85,B 0,C 180,E1 11593.684,E2 11593.684} C_VEL
LIN {X 0,Y 526.14,Z 1114.73,A -85,B 0,C 180,E1 11598.372,E2 11598.372} C_VEL
LIN {X 0,Y 525.389,Z 1124.335,A -85,B 0,C 180,E1 11602.545,E2 11602.545} C_VEL
LIN {X 0,Y 525.179,Z 1129.72,A -85,B 0,C 180,E1 11606.694,E2 11606.694} C_VEL
LIN {X 0,Y 525.254,Z 1130.995,A -85,B 0,C 180,E1 11610.001,E2 11610.001} C_VEL
LIN {X 0,Y 525.246,Z 1127.996,A -85,B 0,C 180,E1 11614.966,E2 11614.966} C_VEL
LIN {X 0,Y 525.665,Z 1120.794,A -85,B 0,C 180,E1 11619.123,E2 11619.123} C_VEL
LIN {X 0,Y 526.678,Z 1109.221,A -85,B 0,C 180,E1 11623.307,E2 11623.307} C_VEL
LIN {X 0,Y 529.008,Z 1090.547,A -85,B 0,C 180,E1 11627.934,E2 11627.934} C_VEL
LIN {X 0,Y 532.911,Z 1065.832,A -85,B 0,C 180,E1 11632.34,E2 11632.34} C_VEL
LIN {X 0,Y 538.161,Z 1036.755,A -85,B 0,C 180,E1 11636.193,E2 11636.193} C_VEL
LIN {X 0,Y 544.275,Z 1002.285,A -85,B 0,C 180,E1 11639.614,E2 11639.614} C_VEL
LIN {X 0,Y 550.382,Z 964.899,A -85,B 0,C 180,E1 11642.362,E2 11642.362} C_VEL
LIN {X 0,Y 555.862,Z 924.407,A -85,B 0,C 180,E1 11644.505,E2 11644.505} C_VEL
LIN {X 0,Y 560.098,Z 881.734,A -85,B 0,C 180,E1 11646.019,E2 11646.019} C_VEL
LIN {X 0,Y 561.444,Z 855.43,A -85,B 0,C 180,E1 11646.654,E2 11646.654} C_VEL
LIN {X 0,Y 537.208,Z 808.148,A -85,B 0,C 180,E1 11649.613,E2 11649.613} C_VEL
LIN {X 0,Y 523.951,Z 784.825,A -85,B 0,C 180,E1 11651.312,E2 11651.312} C_VEL
LIN {X 0,Y 523.789,Z 783.31,A -85,B 0,C 180,E1 11651.36,E2 11651.36} C_VEL
LIN {X 0,Y 523.765,Z 783.31,A -85,B 0,C 180,E1 11656.322,E2 11656.322} C_VEL
LIN {X 0,Y 523.738,Z 783.31,A -85,B 0,C 180,E1 11662.585,E2 11662.585} C_VEL
LIN {X 0,Y 523.923,Z 783.31,A -85,B 0,C 180,E1 11668.627,E2 11668.627} C_VEL
LIN {X 0,Y 524.069,Z 783.31,A -85,B 0,C 180,E1 11674.295,E2 11674.295} C_VEL
LIN {X 0,Y 524.278,Z 783.31,A -85,B 0,C 180,E1 11679.704,E2 11679.704} C_VEL
LIN {X 0,Y 524.393,Z 783.31,A -85,B 0,C 180,E1 11684.922,E2 11684.922} C_VEL
LIN {X 0,Y 524.591,Z 783.31,A -85,B 0,C 180,E1 11690.015,E2 11690.015} C_VEL
LIN {X 0,Y 524.832,Z 783.31,A -85,B 0,C 180,E1 11695.026,E2 11695.026} C_VEL
LIN {X 0,Y 525.015,Z 783.31,A -85,B 0,C 180,E1 11699.994,E2 11699.994} C_VEL
LIN {X 0,Y 524.852,Z 783.31,A -85,B 0,C 180,E1 11704.962,E2 11704.962} C_VEL
LIN {X 0,Y 524.552,Z 783.31,A -85,B 0,C 180,E1 11710.854,E2 11710.854} C_VEL
LIN {X 0,Y 524.411,Z 783.31,A -85,B 0,C 180,E1 11716.786,E2 11716.786} C_VEL
LIN {X 0,Y 524.174,Z 783.31,A -85,B 0,C 180,E1 11722.331,E2 11722.331} C_VEL
LIN {X 0,Y 524.069,Z 783.31,A -85,B 0,C 180,E1 11727.544,E2 11727.544} C_VEL
LIN {X 0,Y 523.922,Z 783.31,A -85,B 0,C 180,E1 11733.32,E2 11733.32} C_VEL
LIN {X 0,Y 523.708,Z 783.31,A -85,B 0,C 180,E1 11739.518,E2 11739.518} C_VEL
LIN {X 0,Y 523.712,Z 783.513,A -85,B 0,C 180,E1 11745.274,E2 11745.274} C_VEL
LIN {X 0,Y 526.197,Z 789.056,A -85,B 0,C 180,E1 11745.63,E2 11745.63} C_VEL
LIN {X 0,Y 550.766,Z 834.62,A -85,B 0,C 180,E1 11748.736,E2 11748.736} C_VEL
LIN {X 0,Y 561.971,Z 862.267,A -85,B 0,C 180,E1 11750.295,E2 11750.295} C_VEL
LIN {X 0,Y 558.116,Z 906.068,A -85,B 0,C 180,E1 11751.57,E2 11751.57} C_VEL
LIN {X 0,Y 553.365,Z 947.238,A -85,B 0,C 180,E1 11753.374,E2 11753.374} C_VEL
LIN {X 0,Y 547.53,Z 989.042,A -85,B 0,C 180,E1 11755.918,E2 11755.918} C_VEL
LIN {X 0,Y 541.327,Z 1028.848,A -85,B 0,C 180,E1 11759.185,E2 11759.185} C_VEL
LIN {X 0,Y 535.784,Z 1063.475,A -85,B 0,C 180,E1 11762.925,E2 11762.925} C_VEL
LIN {X 0,Y 532.979,Z 1081.122,A -85,B 0,C 180,E1 11765.285,E2 11765.285} C_VEL
LIN {X 0,Y 531.033,Z 1086.426,A -85,B 0,C 180,E1 11766.01,E2 11766.01} C_VEL
LIN {X 0,Y 522.665,Z 1100.047,A -85,B 0,C 180,E1 11767.992,E2 11767.992} C_VEL
LIN {X 0,Y 522.423,Z 1101.209,A -85,B 0,C 180,E1 11768.193,E2 11768.193} C_VEL
LIN {X 0,Y 519.651,Z 1122.798,A -85,B 0,C 180,E1 11772.609,E2 11772.609} C_VEL
LIN {X 0,Y 518.102,Z 1139.778,A -85,B 0,C 180,E1 11777.329,E2 11777.329} C_VEL
LIN {X 0,Y 517.468,Z 1150.133,A -85,B 0,C 180,E1 11781.58,E2 11781.58} C_VEL
LIN {X 0,Y 517.334,Z 1155.367,A -85,B 0,C 180,E1 11784.958,E2 11784.958} C_VEL
LIN {X 0,Y 517.274,Z 1158.337,A -85,B 0,C 180,E1 11789.999,E2 11789.999} C_VEL
LIN {X 0,Y 517.308,Z 1155.368,A -85,B 0,C 180,E1 11795.04,E2 11795.04} C_VEL
LIN {X 0,Y 517.543,Z 1148.492,A -85,B 0,C 180,E1 11799.265,E2 11799.265} C_VEL
LIN {X 0,Y 518.528,Z 1134.322,A -85,B 0,C 180,E1 11804.38,E2 11804.38} C_VEL
LIN {X 0,Y 520.63,Z 1114.859,A -85,B 0,C 180,E1 11809.162,E2 11809.162} C_VEL
LIN {X 0,Y 523.846,Z 1091.62,A -85,B 0,C 180,E1 11813.433,E2 11813.433} C_VEL
LIN {X 0,Y 528.546,Z 1062.717,A -85,B 0,C 180,E1 11817.531,E2 11817.531} C_VEL
LIN {X 0,Y 534.6,Z 1026.658,A -85,B 0,C 180,E1 11821.441,E2 11821.441} C_VEL
LIN {X 0,Y 541.091,Z 987.256,A -85,B 0,C 180,E1 11824.664,E2 11824.664} C_VEL
LIN {X 0,Y 547.165,Z 945.176,A -85,B 0,C 180,E1 11827.213,E2 11827.213} C_VEL
LIN {X 0,Y 552.179,Z 903.265,A -85,B 0,C 180,E1 11829.018,E2 11829.018} C_VEL
LIN {X 0,Y 555.168,Z 862.322,A -85,B 0,C 180,E1 11830.257,E2 11830.257} C_VEL
LIN {X 0,Y 539.101,Z 826.343,A -85,B 0,C 180,E1 11832.459,E2 11832.459} C_VEL
LIN {X 0,Y 517.528,Z 788.047,A -85,B 0,C 180,E1 11835.292,E2 11835.292} C_VEL
LIN {X 0,Y 515.912,Z 783.31,A -85,B 0,C 180,E1 11835.638,E2 11835.638} C_VEL
LIN {X 0,Y 515.836,Z 783.31,A -85,B 0,C 180,E1 11841.927,E2 11841.927} C_VEL
LIN {X 0,Y 516.01,Z 783.31,A -85,B 0,C 180,E1 11848.375,E2 11848.375} C_VEL
LIN {X 0,Y 516.203,Z 783.31,A -85,B 0,C 180,E1 11853.888,E2 11853.888} C_VEL
LIN {X 0,Y 516.374,Z 783.31,A -85,B 0,C 180,E1 11859.872,E2 11859.872} C_VEL
LIN {X 0,Y 516.439,Z 783.31,A -85,B 0,C 180,E1 11865.5,E2 11865.5} C_VEL
LIN {X 0,Y 516.744,Z 783.31,A -85,B 0,C 180,E1 11871.577,E2 11871.577} C_VEL
LIN {X 0,Y 516.969,Z 783.31,A -85,B 0,C 180,E1 11876.646,E2 11876.646} C_VEL
LIN {X 0,Y 517.073,Z 783.31,A -85,B 0,C 180,E1 11881.685,E2 11881.685} C_VEL
LIN {X 0,Y 516.832,Z 783.31,A -85,B 0,C 180,E1 11886.74,E2 11886.74} C_VEL
LIN {X 0,Y 516.607,Z 783.31,A -85,B 0,C 180,E1 11891.853,E2 11891.853} C_VEL
LIN {X 0,Y 516.448,Z 783.31,A -85,B 0,C 180,E1 11897.065,E2 11897.065} C_VEL
LIN {X 0,Y 516.232,Z 783.31,A -85,B 0,C 180,E1 11902.435,E2 11902.435} C_VEL
LIN {X 0,Y 516.039,Z 783.31,A -85,B 0,C 180,E1 11908.259,E2 11908.259} C_VEL
LIN {X 0,Y 515.885,Z 783.31,A -85,B 0,C 180,E1 11913.924,E2 11913.924} C_VEL
LIN {X 0,Y 515.835,Z 783.31,A -85,B 0,C 180,E1 11920.26,E2 11920.26} C_VEL
LIN {X 0,Y 515.782,Z 783.31,A -85,B 0,C 180,E1 11925.171,E2 11925.171} C_VEL
LIN {X 0,Y 515.846,Z 783.862,A -85,B 0,C 180,E1 11927.719,E2 11927.719} C_VEL
LIN {X 0,Y 521.078,Z 793.959,A -85,B 0,C 180,E1 11928.451,E2 11928.451} C_VEL
LIN {X 0,Y 545.547,Z 838.238,A -85,B 0,C 180,E1 11931.549,E2 11931.549} C_VEL
LIN {X 0,Y 555.348,Z 860.382,A -85,B 0,C 180,E1 11932.871,E2 11932.871} C_VEL
LIN {X 0,Y 552.167,Z 901.059,A -85,B 0,C 180,E1 11934.001,E2 11934.001} C_VEL
LIN {X 0,Y 547.391,Z 940.383,A -85,B 0,C 180,E1 11935.671,E2 11935.671} C_VEL
LIN {X 0,Y 541.446,Z 979.138,A -85,B 0,C 180,E1 11938.017,E2 11938.017} C_VEL
LIN {X 0,Y 534.899,Z 1016.111,A -85,B 0,C 180,E1 11941.1,E2 11941.1} C_VEL
LIN {X 0,Y 528.752,Z 1048.782,A -85,B 0,C 180,E1 11944.772,E2 11944.772} C_VEL
LIN {X 0,Y 523.946,Z 1075.713,A -85,B 0,C 180,E1 11948.811,E2 11948.811} C_VEL
LIN {X 0,Y 520.401,Z 1098.319,A -85,B 0,C 180,E1 11953.402,E2 11953.402} C_VEL
LIN {X 0,Y 518.318,Z 1114.967,A -85,B 0,C 180,E1 11958.194,E2 11958.194} C_VEL
LIN {X 0,Y 517.515,Z 1124.558,A -85,B 0,C 180,E1 11962.431,E2 11962.431} C_VEL
LIN {X 0,Y 517.279,Z 1129.93,A -85,B 0,C 180,E1 11966.643,E2 11966.643} C_VEL
LIN {X 0,Y 517.356,Z 1131.203,A -85,B 0,C 180,E1 11970.001,E2 11970.001} C_VEL
LIN {X 0,Y 517.365,Z 1128.212,A -85,B 0,C 180,E1 11975.042,E2 11975.042} C_VEL
LIN {X 0,Y 517.801,Z 1121.025,A -85,B 0,C 180,E1 11979.263,E2 11979.263} C_VEL
LIN {X 0,Y 519.073,Z 1107.986,A -85,B 0,C 180,E1 11983.936,E2 11983.936} C_VEL
LIN {X 0,Y 521.516,Z 1089.768,A -85,B 0,C 180,E1 11988.42,E2 11988.42} C_VEL
LIN {X 0,Y 525.677,Z 1065.158,A -85,B 0,C 180,E1 11992.818,E2 11992.818} C_VEL
LIN {X 0,Y 531.142,Z 1035.998,A -85,B 0,C 180,E1 11996.7,E2 11996.7} C_VEL
LIN {X 0,Y 537.399,Z 1002.685,A -85,B 0,C 180,E1 12000.031,E2 12000.031} C_VEL
LIN {X 0,Y 543.737,Z 965.2,A -85,B 0,C 180,E1 12002.82,E2 12002.82} C_VEL
LIN {X 0,Y 549.39,Z 925.036,A -85,B 0,C 180,E1 12004.97,E2 12004.97} C_VEL
LIN {X 0,Y 553.815,Z 882.223,A -85,B 0,C 180,E1 12006.508,E2 12006.508} C_VEL
LIN {X 0,Y 554.974,Z 857.848,A -85,B 0,C 180,E1 12007.126,E2 12007.126} C_VEL
LIN {X 0,Y 531.613,Z 811.921,A -85,B 0,C 180,E1 12010.083,E2 12010.083} C_VEL
LIN {X 0,Y 516.059,Z 785.138,A -85,B 0,C 180,E1 12012.132,E2 12012.132} C_VEL
LIN {X 0,Y 515.83,Z 783.31,A -85,B 0,C 180,E1 12012.333,E2 12012.333} C_VEL
LIN {X 0,Y 515.79,Z 783.31,A -85,B 0,C 180,E1 12017.493,E2 12017.493} C_VEL
LIN {X 0,Y 515.808,Z 783.31,A -85,B 0,C 180,E1 12024.017,E2 12024.017} C_VEL
LIN {X 0,Y 516.039,Z 783.31,A -85,B 0,C 180,E1 12030.052,E2 12030.052} C_VEL
LIN {X 0,Y 516.195,Z 783.31,A -85,B 0,C 180,E1 12035.732,E2 12035.732} C_VEL
LIN {X 0,Y 516.379,Z 783.31,A -85,B 0,C 180,E1 12041.165,E2 12041.165} C_VEL
LIN {X 0,Y 516.506,Z 783.31,A -85,B 0,C 180,E1 12046.422,E2 12046.422} C_VEL
LIN {X 0,Y 516.77,Z 783.31,A -85,B 0,C 180,E1 12052.172,E2 12052.172} C_VEL
LIN {X 0,Y 516.995,Z 783.31,A -85,B 0,C 180,E1 12058.314,E2 12058.314} C_VEL
LIN {X 0,Y 516.955,Z 783.31,A -85,B 0,C 180,E1 12063.354,E2 12063.354} C_VEL
LIN {X 0,Y 516.752,Z 783.31,A -85,B 0,C 180,E1 12068.423,E2 12068.423} C_VEL
LIN {X 0,Y 516.524,Z 783.31,A -85,B 0,C 180,E1 12074.525,E2 12074.525} C_VEL
LIN {X 0,Y 516.33,Z 783.31,A -85,B 0,C 180,E1 12080.609,E2 12080.609} C_VEL
LIN {X 0,Y 516.151,Z 783.31,A -85,B 0,C 180,E1 12086.115,E2 12086.115} C_VEL
LIN {X 0,Y 516.014,Z 783.31,A -85,B 0,C 180,E1 12091.896,E2 12091.896} C_VEL
LIN {X 0,Y 515.813,Z 783.31,A -85,B 0,C 180,E1 12098.075,E2 12098.075} C_VEL
LIN {X 0,Y 515.855,Z 784.091,A -85,B 0,C 180,E1 12104.467,E2 12104.467} C_VEL
LIN {X 0,Y 544.4,Z 836.921,A -85,B 0,C 180,E1 12108.23,E2 12108.23} C_VEL
LIN {X 0,Y 555.614,Z 864.514,A -85,B 0,C 180,E1 12109.844,E2 12109.844} C_VEL
LIN {X 0,Y 551.443,Z 909.48,A -85,B 0,C 180,E1 12111.205,E2 12111.205} C_VEL
LIN {X 0,Y 546.448,Z 950.019,A -85,B 0,C 180,E1 12113.048,E2 12113.048} C_VEL
LIN {X 0,Y 540.805,Z 988.585,A -85,B 0,C 180,E1 12115.433,E2 12115.433} C_VEL
LIN {X 0,Y 534.454,Z 1027.717,A -85,B 0,C 180,E1 12118.662,E2 12118.662} C_VEL
LIN {X 0,Y 528.577,Z 1062.678,A -85,B 0,C 180,E1 12122.468,E2 12122.468} C_VEL
LIN {X 0,Y 523.639,Z 1092.958,A -85,B 0,C 180,E1 12126.78,E2 12126.78} C_VEL
LIN {X 0,Y 522.423,Z 1101.209,A -85,B 0,C 180,E1 12128.193,E2 12128.193} C_VEL
LIN {X 0,Y 517.388,Z 1110.208,A -85,B 0,C 180,E1 12129.758,E2 12129.758} C_VEL
LIN {X 0,Y 512.381,Z 1118.495,A -85,B 0,C 180,E1 12131.392,E2 12131.392} C_VEL
LIN {X 0,Y 510.562,Z 1135.431,A -85,B 0,C 180,E1 12135.827,E2 12135.827} C_VEL
LIN {X 0,Y 509.699,Z 1148.24,A -85,B 0,C 180,E1 12140.589,E2 12140.589} C_VEL
LIN {X 0,Y 509.451,Z 1155.148,A -85,B 0,C 180,E1 12144.88,E2 12144.88} C_VEL
LIN {X 0,Y 509.376,Z 1158.13,A -85,B 0,C 180,E1 12149.999,E2 12149.999} C_VEL
LIN {X 0,Y 509.432,Z 1155.151,A -85,B 0,C 180,E1 12155.118,E2 12155.118} C_VEL
LIN {X 0,Y 509.653,Z 1148.245,A -85,B 0,C 180,E1 12159.409,E2 12159.409} C_VEL
LIN {X 0,Y 510.59,Z 1135.444,A -85,B 0,C 180,E1 12164.169,E2 12164.169} C_VEL
LIN {X 0,Y 512.545,Z 1117.382,A -85,B 0,C 180,E1 12168.849,E2 12168.849} C_VEL
LIN {X 0,Y 515.892,Z 1094.036,A -85,B 0,C 180,E1 12173.357,E2 12173.357} C_VEL
LIN {X 0,Y 521.001,Z 1064.114,A -85,B 0,C 180,E1 12177.729,E2 12177.729} C_VEL
LIN {X 0,Y 527.303,Z 1028.266,A -85,B 0,C 180,E1 12181.714,E2 12181.714} C_VEL
LIN {X 0,Y 533.89,Z 989.668,A -85,B 0,C 180,E1 12184.952,E2 12184.952} C_VEL
LIN {X 0,Y 539.835,Z 951.176,A -85,B 0,C 180,E1 12187.376,E2 12187.376} C_VEL
LIN {X 0,Y 545.1,Z 910.047,A -85,B 0,C 180,E1 12189.279,E2 12189.279} C_VEL
LIN {X 0,Y 548.664,Z 864.39,A -85,B 0,C 180,E1 12190.743,E2 12190.743} C_VEL
LIN {X 0,Y 533.052,Z 829.321,A -85,B 0,C 180,E1 12192.967,E2 12192.967} C_VEL
LIN {X 0,Y 510.471,Z 789.045,A -85,B 0,C 180,E1 12196.03,E2 12196.03} C_VEL
LIN {X 0,Y 508.008,Z 783.31,A -85,B 0,C 180,E1 12196.433,E2 12196.433} C_VEL
LIN {X 0,Y 507.928,Z 783.31,A -85,B 0,C 180,E1 12203.385,E2 12203.385} C_VEL
LIN {X 0,Y 508.132,Z 783.31,A -85,B 0,C 180,E1 12209.849,E2 12209.849} C_VEL
LIN {X 0,Y 508.332,Z 783.31,A -85,B 0,C 180,E1 12215.346,E2 12215.346} C_VEL
LIN {X 0,Y 508.454,Z 783.31,A -85,B 0,C 180,E1 12220.874,E2 12220.874} C_VEL
LIN {X 0,Y 508.576,Z 783.31,A -85,B 0,C 180,E1 12226.219,E2 12226.219} C_VEL
LIN {X 0,Y 508.82,Z 783.31,A -85,B 0,C 180,E1 12231.445,E2 12231.445} C_VEL
LIN {X 0,Y 509.078,Z 783.31,A -85,B 0,C 180,E1 12236.594,E2 12236.594} C_VEL
LIN {X 0,Y 509.178,Z 783.31,A -85,B 0,C 180,E1 12241.711,E2 12241.711} C_VEL
LIN {X 0,Y 508.913,Z 783.31,A -85,B 0,C 180,E1 12246.845,E2 12246.845} C_VEL
LIN {X 0,Y 508.689,Z 783.31,A -85,B 0,C 180,E1 12252.04,E2 12252.04} C_VEL
LIN {X 0,Y 508.476,Z 783.31,A -85,B 0,C 180,E1 12257.539,E2 12257.539} C_VEL
LIN {X 0,Y 508.272,Z 783.31,A -85,B 0,C 180,E1 12262.806,E2 12262.806} C_VEL
LIN {X 0,Y 508.128,Z 783.31,A -85,B 0,C 180,E1 12268.5,E2 12268.5} C_VEL
LIN {X 0,Y 507.986,Z 783.31,A -85,B 0,C 180,E1 12274.525,E2 12274.525} C_VEL
LIN {X 0,Y 507.837,Z 783.31,A -85,B 0,C 180,E1 12281.028,E2 12281.028} C_VEL
LIN {X 0,Y 507.848,Z 783.31,A -85,B 0,C 180,E1 12286.807,E2 12286.807} C_VEL
LIN {X 0,Y 510.331,Z 789.031,A -85,B 0,C 180,E1 12287.214,E2 12287.214} C_VEL
LIN {X 0,Y 535.702,Z 833.648,A -85,B 0,C 180,E1 12290.571,E2 12290.571} C_VEL
LIN {X 0,Y 549.031,Z 861.622,A -85,B 0,C 180,E1 12292.369,E2 12292.369} C_VEL
LIN {X 0,Y 545.575,Z 903.783,A -85,B 0,C 180,E1 12293.585,E2 12293.585} C_VEL
LIN {X 0,Y 540.625,Z 942.781,A -85,B 0,C 180,E1 12295.302,E2 12295.302} C_VEL
LIN {X 0,Y 534.577,Z 980.304,A -85,B 0,C 180,E1 12297.623,E2 12297.623} C_VEL
LIN {X 0,Y 527.925,Z 1016.452,A -85,B 0,C 180,E1 12300.681,E2 12300.681} C_VEL
LIN {X 0,Y 521.523,Z 1048.824,A -85,B 0,C 180,E1 12304.359,E2 12304.359} C_VEL
LIN {X 0,Y 516.417,Z 1075.989,A -85,B 0,C 180,E1 12308.486,E2 12308.486} C_VEL
LIN {X 0,Y 512.738,Z 1098.283,A -85,B 0,C 180,E1 12313.072,E2 12313.072} C_VEL
LIN {X 0,Y 510.494,Z 1115.199,A -85,B 0,C 180,E1 12318.01,E2 12318.01} C_VEL
LIN {X 0,Y 509.665,Z 1124.777,A -85,B 0,C 180,E1 12322.313,E2 12322.313} C_VEL
LIN {X 0,Y 509.406,Z 1130.138,A -85,B 0,C 180,E1 12326.591,E2 12326.591} C_VEL
LIN {X 0,Y 509.458,Z 1131.41,A -85,B 0,C 180,E1 12330.001,E2 12330.001} C_VEL
LIN {X 0,Y 509.484,Z 1128.425,A -85,B 0,C 180,E1 12335.12,E2 12335.12} C_VEL
LIN {X 0,Y 509.951,Z 1121.252,A -85,B 0,C 180,E1 12339.407,E2 12339.407} C_VEL
LIN {X 0,Y 511.306,Z 1108.232,A -85,B 0,C 180,E1 12344.152,E2 12344.152} C_VEL
LIN {X 0,Y 513.91,Z 1090.038,A -85,B 0,C 180,E1 12348.702,E2 12348.702} C_VEL
LIN {X 0,Y 518.112,Z 1066.355,A -85,B 0,C 180,E1 12353.027,E2 12353.027} C_VEL
LIN {X 0,Y 524.004,Z 1036.338,A -85,B 0,C 180,E1 12357.093,E2 12357.093} C_VEL
LIN {X 0,Y 530.538,Z 1003.076,A -85,B 0,C 180,E1 12360.461,E2 12360.461} C_VEL
LIN {X 0,Y 537.195,Z 965.008,A -85,B 0,C 180,E1 12363.32,E2 12363.32} C_VEL
LIN {X 0,Y 543.097,Z 924.527,A -85,B 0,C 180,E1 12365.497,E2 12365.497} C_VEL
LIN {X 0,Y 547.654,Z 881.833,A -85,B 0,C 180,E1 12367.035,E2 12367.035} C_VEL
LIN {X 0,Y 548.822,Z 860.867,A -85,B 0,C 180,E1 12367.571,E2 12367.571} C_VEL
LIN {X 0,Y 526.361,Z 816.276,A -85,B 0,C 180,E1 12370.522,E2 12370.522} C_VEL
LIN {X 0,Y 508.037,Z 784.899,A -85,B 0,C 180,E1 12373.013,E2 12373.013} C_VEL
LIN {X 0,Y 507.874,Z 783.31,A -85,B 0,C 180,E1 12373.195,E2 12373.195} C_VEL
LIN {X 0,Y 507.808,Z 783.31,A -85,B 0,C 180,E1 12378.969,E2 12378.969} C_VEL
LIN {X 0,Y 507.901,Z 783.31,A -85,B 0,C 180,E1 12385.468,E2 12385.468} C_VEL
LIN {X 0,Y 508.159,Z 783.31,A -85,B 0,C 180,E1 12391.502,E2 12391.502} C_VEL
LIN {X 0,Y 508.363,Z 783.31,A -85,B 0,C 180,E1 12397.514,E2 12397.514} C_VEL
LIN {X 0,Y 508.502,Z 783.31,A -85,B 0,C 180,E1 12402.659,E2 12402.659} C_VEL
LIN {X 0,Y 508.677,Z 783.31,A -85,B 0,C 180,E1 12407.96,E2 12407.96} C_VEL
LIN {X 0,Y 508.946,Z 783.31,A -85,B 0,C 180,E1 12413.155,E2 12413.155} C_VEL
LIN {X 0,Y 509.107,Z 783.31,A -85,B 0,C 180,E1 12418.288,E2 12418.288} C_VEL
LIN {X 0,Y 509.069,Z 783.31,A -85,B 0,C 180,E1 12423.406,E2 12423.406} C_VEL
LIN {X 0,Y 508.832,Z 783.31,A -85,B 0,C 180,E1 12428.555,E2 12428.555} C_VEL
LIN {X 0,Y 508.657,Z 783.31,A -85,B 0,C 180,E1 12433.778,E2 12433.778} C_VEL
LIN {X 0,Y 508.471,Z 783.31,A -85,B 0,C 180,E1 12439.126,E2 12439.126} C_VEL
LIN {X 0,Y 508.245,Z 783.31,A -85,B 0,C 180,E1 12444.659,E2 12444.659} C_VEL
LIN {X 0,Y 508.123,Z 783.31,A -85,B 0,C 180,E1 12450.448,E2 12450.448} C_VEL
LIN {X 0,Y 507.921,Z 783.31,A -85,B 0,C 180,E1 12456.616,E2 12456.616} C_VEL
LIN {X 0,Y 507.918,Z 783.78,A -85,B 0,C 180,E1 12463.596,E2 12463.596} C_VEL
LIN {X 0,Y 510.659,Z 789.305,A -85,B 0,C 180,E1 12464.01,E2 12464.01} C_VEL
LIN {X 0,Y 536.057,Z 835.411,A -85,B 0,C 180,E1 12467.445,E2 12467.445} C_VEL
LIN {X 0,Y 549.181,Z 866.065,A -85,B 0,C 180,E1 12469.361,E2 12469.361} C_VEL
LIN {X 0,Y 544.861,Z 911.844,A -85,B 0,C 180,E1 12470.789,E2 12470.789} C_VEL
LIN {X 0,Y 539.197,Z 955.312,A -85,B 0,C 180,E1 12472.849,E2 12472.849} C_VEL
LIN {X 0,Y 532.975,Z 994.987,A -85,B 0,C 180,E1 12475.451,E2 12475.451} C_VEL
LIN {X 0,Y 526.854,Z 1030.728,A -85,B 0,C 180,E1 12478.537,E2 12478.537} C_VEL
LIN {X 0,Y 521.013,Z 1064.073,A -85,B 0,C 180,E1 12482.269,E2 12482.269} C_VEL
LIN {X 0,Y 515.912,Z 1094.009,A -85,B 0,C 180,E1 12486.64,E2 12486.64} C_VEL
LIN {X 0,Y 512.381,Z 1118.495,A -85,B 0,C 180,E1 12491.392,E2 12491.392} C_VEL
LIN {X 0,Y 507.655,Z 1126.091,A -85,B 0,C 180,E1 12493.087,E2 12493.087} C_VEL
LIN {X 0,Y 503.04,Z 1132.777,A -85,B 0,C 180,E1 12494.857,E2 12494.857} C_VEL
LIN {X 0,Y 501.946,Z 1146.014,A -85,B 0,C 180,E1 12499.564,E2 12499.564} C_VEL
LIN {X 0,Y 501.542,Z 1153.884,A -85,B 0,C 180,E1 12503.929,E2 12503.929} C_VEL
LIN {X 0,Y 501.419,Z 1157.573,A -85,B 0,C 180,E1 12508.267,E2 12508.267} C_VEL
LIN {X 0,Y 501.412,Z 1157.574,A -85,B 0,C 180,E1 12511.73,E2 12511.73} C_VEL
LIN {X 0,Y 501.53,Z 1153.889,A -85,B 0,C 180,E1 12516.068,E2 12516.068} C_VEL
LIN {X 0,Y 502.026,Z 1144.722,A -85,B 0,C 180,E1 12521.005,E2 12521.005} C_VEL
LIN {X 0,Y 503.277,Z 1130.723,A -85,B 0,C 180,E1 12525.719,E2 12525.719} C_VEL
LIN {X 0,Y 505.891,Z 1110.368,A -85,B 0,C 180,E1 12530.603,E2 12530.603} C_VEL
LIN {X 0,Y 510.055,Z 1084.494,A -85,B 0,C 180,E1 12535.225,E2 12535.225} C_VEL
LIN {X 0,Y 515.986,Z 1051.223,A -85,B 0,C 180,E1 12539.703,E2 12539.703} C_VEL
LIN {X 0,Y 522.95,Z 1013.737,A -85,B 0,C 180,E1 12543.498,E2 12543.498} C_VEL
LIN {X 0,Y 530.042,Z 972.264,A -85,B 0,C 180,E1 12546.634,E2 12546.634} C_VEL
LIN {X 0,Y 536.54,Z 927.973,A -85,B 0,C 180,E1 12549.051,E2 12549.051} C_VEL
LIN {X 0,Y 541.865,Z 880.84,A -85,B 0,C 180,E1 12550.779,E2 12550.779} C_VEL
LIN {X 0,Y 542.336,Z 866.957,A -85,B 0,C 180,E1 12551.202,E2 12551.202} C_VEL
LIN {X 0,Y 526.147,Z 830.544,A -85,B 0,C 180,E1 12553.606,E2 12553.606} C_VEL
LIN {X 0,Y 505.049,Z 793.446,A -85,B 0,C 180,E1 12556.545,E2 12556.545} C_VEL
LIN {X 0,Y 500.077,Z 784.522,A -85,B 0,C 180,E1 12557.3,E2 12557.3} C_VEL
LIN {X 0,Y 499.951,Z 783.31,A -85,B 0,C 180,E1 12557.422,E2 12557.422} C_VEL
LIN {X 0,Y 499.926,Z 783.31,A -85,B 0,C 180,E1 12562.7,E2 12562.7} C_VEL
LIN {X 0,Y 500.113,Z 783.31,A -85,B 0,C 180,E1 12569.011,E2 12569.011} C_VEL
LIN {X 0,Y 500.445,Z 783.31,A -85,B 0,C 180,E1 12575.266,E2 12575.266} C_VEL
LIN {X 0,Y 500.506,Z 783.31,A -85,B 0,C 180,E1 12580.558,E2 12580.558} C_VEL
LIN {X 0,Y 500.641,Z 783.31,A -85,B 0,C 180,E1 12585.997,E2 12585.997} C_VEL
LIN {X 0,Y 500.926,Z 783.31,A -85,B 0,C 180,E1 12591.309,E2 12591.309} C_VEL
LIN {X 0,Y 501.168,Z 783.31,A -85,B 0,C 180,E1 12596.54,E2 12596.54} C_VEL
LIN {X 0,Y 501.271,Z 783.31,A -85,B 0,C 180,E1 12601.738,E2 12601.738} C_VEL
LIN {X 0,Y 501.023,Z 783.31,A -85,B 0,C 180,E1 12606.954,E2 12606.954} C_VEL
LIN {X 0,Y 500.76,Z 783.31,A -85,B 0,C 180,E1 12612.233,E2 12612.233} C_VEL
LIN {X 0,Y 500.575,Z 783.31,A -85,B 0,C 180,E1 12617.624,E2 12617.624} C_VEL
LIN {X 0,Y 500.313,Z 783.31,A -85,B 0,C 180,E1 12623.189,E2 12623.189} C_VEL
LIN {X 0,Y 500.187,Z 783.31,A -85,B 0,C 180,E1 12628.995,E2 12628.995} C_VEL
LIN {X 0,Y 500.029,Z 783.31,A -85,B 0,C 180,E1 12635.155,E2 12635.155} C_VEL
LIN {X 0,Y 499.956,Z 783.31,A -85,B 0,C 180,E1 12641.819,E2 12641.819} C_VEL
LIN {X 0,Y 499.929,Z 783.449,A -85,B 0,C 180,E1 12645.923,E2 12645.923} C_VEL
LIN {X 0,Y 502.388,Z 789.038,A -85,B 0,C 180,E1 12646.317,E2 12646.317} C_VEL
LIN {X 0,Y 526.912,Z 831.467,A -85,B 0,C 180,E1 12649.693,E2 12649.693} C_VEL
LIN {X 0,Y 542.772,Z 864.524,A -85,B 0,C 180,E1 12651.9,E2 12651.9} C_VEL
LIN {X 0,Y 538.709,Z 909.122,A -85,B 0,C 180,E1 12653.252,E2 12653.252} C_VEL
LIN {X 0,Y 533.016,Z 950.826,A -85,B 0,C 180,E1 12655.231,E2 12655.231} C_VEL
LIN {X 0,Y 526.466,Z 988.293,A -85,B 0,C 180,E1 12657.738,E2 12657.738} C_VEL
LIN {X 0,Y 519.815,Z 1022.266,A -85,B 0,C 180,E1 12660.814,E2 12660.814} C_VEL
LIN {X 0,Y 513.691,Z 1051.923,A -85,B 0,C 180,E1 12664.359,E2 12664.359} C_VEL
LIN {X 0,Y 508.698,Z 1077.427,A -85,B 0,C 180,E1 12668.373,E2 12668.373} C_VEL
LIN {X 0,Y 504.954,Z 1099.157,A -85,B 0,C 180,E1 12672.97,E2 12672.97} C_VEL
LIN {X 0,Y 502.675,Z 1115.428,A -85,B 0,C 180,E1 12677.821,E2 12677.821} C_VEL
LIN {X 0,Y 501.805,Z 1124.994,A -85,B 0,C 180,E1 12682.192,E2 12682.192} C_VEL
LIN {X 0,Y 501.506,Z 1130.347,A -85,B 0,C 180,E1 12686.537,E2 12686.537} C_VEL
LIN {X 0,Y 501.56,Z 1131.617,A -85,B 0,C 180,E1 12690.002,E2 12690.002} C_VEL
LIN {X 0,Y 501.612,Z 1128.637,A -85,B 0,C 180,E1 12695.201,E2 12695.201} C_VEL
LIN {X 0,Y 502.099,Z 1121.476,A -85,B 0,C 180,E1 12699.555,E2 12699.555} C_VEL
LIN {X 0,Y 503.545,Z 1108.474,A -85,B 0,C 180,E1 12704.375,E2 12704.375} C_VEL
LIN {X 0,Y 506.302,Z 1090.302,A -85,B 0,C 180,E1 12708.994,E2 12708.994} C_VEL
LIN {X 0,Y 510.807,Z 1066.267,A -85,B 0,C 180,E1 12713.437,E2 12713.437} C_VEL
LIN {X 0,Y 516.877,Z 1036.663,A -85,B 0,C 180,E1 12717.498,E2 12717.498} C_VEL
LIN {X 0,Y 523.666,Z 1003.462,A -85,B 0,C 180,E1 12720.904,E2 12720.904} C_VEL
LIN {X 0,Y 530.483,Z 966.23,A -85,B 0,C 180,E1 12723.741,E2 12723.741} C_VEL
LIN {X 0,Y 536.549,Z 926.203,A -85,B 0,C 180,E1 12725.935,E2 12725.935} C_VEL
LIN {X 0,Y 541.312,Z 883.635,A -85,B 0,C 180,E1 12727.507,E2 12727.507} C_VEL
LIN {X 0,Y 542.511,Z 863.54,A -85,B 0,C 180,E1 12728.051,E2 12728.051} C_VEL
LIN {X 0,Y 520.832,Z 820.097,A -85,B 0,C 180,E1 12731.01,E2 12731.01} C_VEL
LIN {X 0,Y 500.089,Z 784.791,A -85,B 0,C 180,E1 12733.925,E2 12733.925} C_VEL
LIN {X 0,Y 499.935,Z 783.31,A -85,B 0,C 180,E1 12734.021,E2 12734.021} C_VEL
LIN {X 0,Y 499.894,Z 783.31,A -85,B 0,C 180,E1 12740.464,E2 12740.464} C_VEL
LIN {X 0,Y 500.057,Z 783.31,A -85,B 0,C 180,E1 12746.944,E2 12746.944} C_VEL
LIN {X 0,Y 500.232,Z 783.31,A -85,B 0,C 180,E1 12752.973,E2 12752.973} C_VEL
LIN {X 0,Y 500.484,Z 783.31,A -85,B 0,C 180,E1 12758.693,E2 12758.693} C_VEL
LIN {X 0,Y 500.621,Z 783.31,A -85,B 0,C 180,E1 12764.188,E2 12764.188} C_VEL
LIN {X 0,Y 500.86,Z 783.31,A -85,B 0,C 180,E1 12769.537,E2 12769.537} C_VEL
LIN {X 0,Y 501.117,Z 783.31,A -85,B 0,C 180,E1 12774.79,E2 12774.79} C_VEL
LIN {X 0,Y 501.314,Z 783.31,A -85,B 0,C 180,E1 12779.994,E2 12779.994} C_VEL
LIN {X 0,Y 501.135,Z 783.31,A -85,B 0,C 180,E1 12785.197,E2 12785.197} C_VEL
LIN {X 0,Y 500.863,Z 783.31,A -85,B 0,C 180,E1 12790.45,E2 12790.45} C_VEL
LIN {X 0,Y 500.677,Z 783.31,A -85,B 0,C 180,E1 12795.797,E2 12795.797} C_VEL
LIN {X 0,Y 500.48,Z 783.31,A -85,B 0,C 180,E1 12801.293,E2 12801.293} C_VEL
LIN {X 0,Y 500.285,Z 783.31,A -85,B 0,C 180,E1 12807.009,E2 12807.009} C_VEL
LIN {X 0,Y 500.096,Z 783.31,A -85,B 0,C 180,E1 12813.038,E2 12813.038} C_VEL
LIN {X 0,Y 499.878,Z 783.31,A -85,B 0,C 180,E1 12819.52,E2 12819.52} C_VEL
LIN {X 0,Y 499.914,Z 783.31,A -85,B 0,C 180,E1 12822.654,E2 12822.654} C_VEL
LIN {X 0,Y 502.369,Z 789.002,A -85,B 0,C 180,E1 12823.075,E2 12823.075} C_VEL
LIN {X 0,Y 526.079,Z 830.62,A -85,B 0,C 180,E1 12826.399,E2 12826.399} C_VEL
LIN {X 0,Y 541.795,Z 865.545,A -85,B 0,C 180,E1 12828.712,E2 12828.712} C_VEL
LIN {X 0,Y 542.662,Z 871.814,A -85,B 0,C 180,E1 12828.995,E2 12828.995} C_VEL
LIN {X 0,Y 538.337,Z 913.878,A -85,B 0,C 180,E1 12830.361,E2 12830.361} C_VEL
LIN {X 0,Y 532.537,Z 956.421,A -85,B 0,C 180,E1 12832.414,E2 12832.414} C_VEL
LIN {X 0,Y 525.693,Z 998.078,A -85,B 0,C 180,E1 12835.215,E2 12835.215} C_VEL
LIN {X 0,Y 519.001,Z 1035.058,A -85,B 0,C 180,E1 12838.543,E2 12838.543} C_VEL
LIN {X 0,Y 512.991,Z 1067.612,A -85,B 0,C 180,E1 12842.36,E2 12842.36} C_VEL
LIN {X 0,Y 508.005,Z 1096.241,A -85,B 0,C 180,E1 12846.721,E2 12846.721} C_VEL
LIN {X 0,Y 504.481,Z 1119.757,A -85,B 0,C 180,E1 12851.44,E2 12851.44} C_VEL
LIN {X 0,Y 503.04,Z 1132.777,A -85,B 0,C 180,E1 12854.857,E2 12854.857} C_VEL
LIN {X 0,Y 498.493,Z 1138.745,A -85,B 0,C 180,E1 12856.674,E2 12856.674} C_VEL
LIN {X 0,Y 494.214,Z 1143.851,A -85,B 0,C 180,E1 12858.551,E2 12858.551} C_VEL
LIN {X 0,Y 493.655,Z 1153.667,A -85,B 0,C 180,E1 12863.832,E2 12863.832} C_VEL
LIN {X 0,Y 493.545,Z 1157.366,A -85,B 0,C 180,E1 12868.239,E2 12868.239} C_VEL
LIN {X 0,Y 493.539,Z 1157.367,A -85,B 0,C 180,E1 12871.758,E2 12871.758} C_VEL
LIN {X 0,Y 493.641,Z 1153.673,A -85,B 0,C 180,E1 12876.166,E2 12876.166} C_VEL
LIN {X 0,Y 494.153,Z 1144.465,A -85,B 0,C 180,E1 12881.195,E2 12881.195} C_VEL
LIN {X 0,Y 495.474,Z 1130.473,A -85,B 0,C 180,E1 12885.974,E2 12885.974} C_VEL
LIN {X 0,Y 498.267,Z 1110.095,A -85,B 0,C 180,E1 12890.933,E2 12890.933} C_VEL
LIN {X 0,Y 502.74,Z 1083.735,A -85,B 0,C 180,E1 12895.693,E2 12895.693} C_VEL
LIN {X 0,Y 508.759,Z 1051.536,A -85,B 0,C 180,E1 12900.086,E2 12900.086} C_VEL
LIN {X 0,Y 516,Z 1014.353,A -85,B 0,C 180,E1 12903.91,E2 12903.91} C_VEL
LIN {X 0,Y 523.428,Z 972.504,A -85,B 0,C 180,E1 12907.12,E2 12907.12} C_VEL
LIN {X 0,Y 530.103,Z 928.843,A -85,B 0,C 180,E1 12909.53,E2 12909.53} C_VEL
LIN {X 0,Y 535.501,Z 882.79,A -85,B 0,C 180,E1 12911.254,E2 12911.254} C_VEL
LIN {X 0,Y 535.935,Z 869.208,A -85,B 0,C 180,E1 12911.691,E2 12911.691} C_VEL
LIN {X 0,Y 519.984,Z 833.245,A -85,B 0,C 180,E1 12914.162,E2 12914.162} C_VEL
LIN {X 0,Y 498.155,Z 794.887,A -85,B 0,C 180,E1 12917.309,E2 12917.309} C_VEL
LIN {X 0,Y 492.173,Z 784.733,A -85,B 0,C 180,E1 12918.244,E2 12918.244} C_VEL
LIN {X 0,Y 492.023,Z 783.31,A -85,B 0,C 180,E1 12918.465,E2 12918.465} C_VEL
LIN {X 0,Y 492.018,Z 783.31,A -85,B 0,C 180,E1 12924.202,E2 12924.202} C_VEL
LIN {X 0,Y 492.251,Z 783.31,A -85,B 0,C 180,E1 12930.507,E2 12930.507} C_VEL
LIN {X 0,Y 492.488,Z 783.31,A -85,B 0,C 180,E1 12936.434,E2 12936.434} C_VEL
LIN {X 0,Y 492.675,Z 783.31,A -85,B 0,C 180,E1 12942.428,E2 12942.428} C_VEL
LIN {X 0,Y 492.778,Z 783.31,A -85,B 0,C 180,E1 12947.579,E2 12947.579} C_VEL
LIN {X 0,Y 493.092,Z 783.31,A -85,B 0,C 180,E1 12952.947,E2 12952.947} C_VEL
LIN {X 0,Y 493.293,Z 783.31,A -85,B 0,C 180,E1 12958.247,E2 12958.247} C_VEL
LIN {X 0,Y 493.277,Z 783.31,A -85,B 0,C 180,E1 12963.528,E2 12963.528} C_VEL
LIN {X 0,Y 492.973,Z 783.31,A -85,B 0,C 180,E1 12968.846,E2 12968.846} C_VEL
LIN {X 0,Y 492.798,Z 783.31,A -85,B 0,C 180,E1 12974.245,E2 12974.245} C_VEL
LIN {X 0,Y 492.552,Z 783.31,A -85,B 0,C 180,E1 12979.783,E2 12979.783} C_VEL
LIN {X 0,Y 492.296,Z 783.31,A -85,B 0,C 180,E1 12985.528,E2 12985.528} C_VEL
LIN {X 0,Y 492.162,Z 783.31,A -85,B 0,C 180,E1 12991.562,E2 12991.562} C_VEL
LIN {X 0,Y 492.03,Z 783.31,A -85,B 0,C 180,E1 12998.02,E2 12998.02} C_VEL
LIN {X 0,Y 492.036,Z 783.31,A -85,B 0,C 180,E1 13002.65,E2 13002.65} C_VEL
LIN {X 0,Y 492.011,Z 783.602,A -85,B 0,C 180,E1 13004.971,E2 13004.971} C_VEL
LIN {X 0,Y 494.454,Z 789.039,A -85,B 0,C 180,E1 13005.378,E2 13005.378} C_VEL
LIN {X 0,Y 518.757,Z 830.278,A -85,B 0,C 180,E1 13008.855,E2 13008.855} C_VEL
LIN {X 0,Y 536.55,Z 867.283,A -85,B 0,C 180,E1 13011.423,E2 13011.423} C_VEL
LIN {X 0,Y 532.196,Z 911.75,A -85,B 0,C 180,E1 13012.823,E2 13012.823} C_VEL
LIN {X 0,Y 526.238,Z 953.152,A -85,B 0,C 180,E1 13014.843,E2 13014.843} C_VEL
LIN {X 0,Y 519.125,Z 992.154,A -85,B 0,C 180,E1 13017.543,E2 13017.543} C_VEL
LIN {X 0,Y 511.969,Z 1027.025,A -85,B 0,C 180,E1 13020.846,E2 13020.846} C_VEL
LIN {X 0,Y 505.269,Z 1058.145,A -85,B 0,C 180,E1 13024.805,E2 13024.805} C_VEL
LIN {X 0,Y 499.86,Z 1084.585,A -85,B 0,C 180,E1 13029.352,E2 13029.352} C_VEL
LIN {X 0,Y 496.404,Z 1104.539,A -85,B 0,C 180,E1 13034.057,E2 13034.057} C_VEL
LIN {X 0,Y 494.599,Z 1118.114,A -85,B 0,C 180,E1 13038.613,E2 13038.613} C_VEL
LIN {X 0,Y 493.811,Z 1126.663,A -85,B 0,C 180,E1 13042.952,E2 13042.952} C_VEL
LIN {X 0,Y 493.578,Z 1131.516,A -85,B 0,C 180,E1 13048.242,E2 13048.242} C_VEL
LIN {X 0,Y 493.655,Z 1131.486,A -85,B 0,C 180,E1 13051.76,E2 13051.76} C_VEL
LIN {X 0,Y 493.855,Z 1126.535,A -85,B 0,C 180,E1 13057.051,E2 13057.051} C_VEL
LIN {X 0,Y 494.896,Z 1115.405,A -85,B 0,C 180,E1 13062.377,E2 13062.377} C_VEL
LIN {X 0,Y 497.24,Z 1099.125,A -85,B 0,C 180,E1 13067.285,E2 13067.285} C_VEL
LIN {X 0,Y 501.496,Z 1076.022,A -85,B 0,C 180,E1 13072.19,E2 13072.19} C_VEL
LIN {X 0,Y 507.592,Z 1047.37,A -85,B 0,C 180,E1 13076.601,E2 13076.601} C_VEL
LIN {X 0,Y 514.459,Z 1015.183,A -85,B 0,C 180,E1 13080.29,E2 13080.29} C_VEL
LIN {X 0,Y 521.673,Z 978.981,A -85,B 0,C 180,E1 13083.372,E2 13083.372} C_VEL
LIN {X 0,Y 528.191,Z 940.395,A -85,B 0,C 180,E1 13085.768,E2 13085.768} C_VEL
LIN {X 0,Y 533.713,Z 898.071,A -85,B 0,C 180,E1 13087.589,E2 13087.589} C_VEL
LIN {X 0,Y 536.163,Z 866.149,A -85,B 0,C 180,E1 13088.549,E2 13088.549} C_VEL
LIN {X 0,Y 515.94,Z 825.075,A -85,B 0,C 180,E1 13091.425,E2 13091.425} C_VEL
LIN {X 0,Y 493.839,Z 788.371,A -85,B 0,C 180,E1 13094.601,E2 13094.601} C_VEL
LIN {X 0,Y 492.02,Z 783.31,A -85,B 0,C 180,E1 13095.032,E2 13095.032} C_VEL
LIN {X 0,Y 491.985,Z 783.31,A -85,B 0,C 180,E1 13100.349,E2 13100.349} C_VEL
LIN {X 0,Y 492.057,Z 783.31,A -85,B 0,C 180,E1 13106.336,E2 13106.336} C_VEL
LIN {X 0,Y 492.311,Z 783.31,A -85,B 0,C 180,E1 13112.502,E2 13112.502} C_VEL
LIN {X 0,Y 492.52,Z 783.31,A -85,B 0,C 180,E1 13118.331,E2 13118.331} C_VEL
LIN {X 0,Y 492.684,Z 783.31,A -85,B 0,C 180,E1 13123.927,E2 13123.927} C_VEL
LIN {X 0,Y 492.969,Z 783.31,A -85,B 0,C 180,E1 13129.596,E2 13129.596} C_VEL
LIN {X 0,Y 493.203,Z 783.31,A -85,B 0,C 180,E1 13134.706,E2 13134.706} C_VEL
LIN {X 0,Y 493.441,Z 783.31,A -85,B 0,C 180,E1 13139.993,E2 13139.993} C_VEL
LIN {X 0,Y 493.218,Z 783.31,A -85,B 0,C 180,E1 13145.281,E2 13145.281} C_VEL
LIN {X 0,Y 492.949,Z 783.31,A -85,B 0,C 180,E1 13150.62,E2 13150.62} C_VEL
LIN {X 0,Y 492.736,Z 783.31,A -85,B 0,C 180,E1 13156.058,E2 13156.058} C_VEL
LIN {X 0,Y 492.519,Z 783.31,A -85,B 0,C 180,E1 13161.655,E2 13161.655} C_VEL
LIN {X 0,Y 492.38,Z 783.31,A -85,B 0,C 180,E1 13167.479,E2 13167.479} C_VEL
LIN {X 0,Y 492.103,Z 783.31,A -85,B 0,C 180,E1 13173.763,E2 13173.763} C_VEL
LIN {X 0,Y 491.963,Z 783.31,A -85,B 0,C 180,E1 13180.285,E2 13180.285} C_VEL
LIN {X 0,Y 492.008,Z 783.31,A -85,B 0,C 180,E1 13181.71,E2 13181.71} C_VEL
LIN {X 0,Y 494.487,Z 789.084,A -85,B 0,C 180,E1 13182.149,E2 13182.149} C_VEL
LIN {X 0,Y 518.243,Z 830.091,A -85,B 0,C 180,E1 13185.608,E2 13185.608} C_VEL
LIN {X 0,Y 534.431,Z 865.307,A -85,B 0,C 180,E1 13188.049,E2 13188.049} C_VEL
LIN {X 0,Y 536.53,Z 871.91,A -85,B 0,C 180,E1 13188.462,E2 13188.462} C_VEL
LIN {X 0,Y 532.064,Z 914.032,A -85,B 0,C 180,E1 13189.842,E2 13189.842} C_VEL
LIN {X 0,Y 525.88,Z 957.797,A -85,B 0,C 180,E1 13191.984,E2 13191.984} C_VEL
LIN {X 0,Y 518.648,Z 999.779,A -85,B 0,C 180,E1 13194.865,E2 13194.865} C_VEL
LIN {X 0,Y 511.451,Z 1037.928,A -85,B 0,C 180,E1 13198.399,E2 13198.399} C_VEL
LIN {X 0,Y 504.892,Z 1071.442,A -85,B 0,C 180,E1 13202.493,E2 13202.493} C_VEL
LIN {X 0,Y 500.074,Z 1098.431,A -85,B 0,C 180,E1 13206.802,E2 13206.802} C_VEL
LIN {X 0,Y 496.721,Z 1119.882,A -85,B 0,C 180,E1 13211.236,E2 13211.236} C_VEL
LIN {X 0,Y 494.669,Z 1137.699,A -85,B 0,C 180,E1 13216.266,E2 13216.266} C_VEL
LIN {X 0,Y 494.214,Z 1143.851,A -85,B 0,C 180,E1 13218.551,E2 13218.551} C_VEL
LIN {X 0,Y 491.495,Z 1147.193,A -85,B 0,C 180,E1 13219.995,E2 13219.995} C_VEL
LIN {X 0,Y 485.858,Z 1151.469,A -85,B 0,C 180,E1 13222.31,E2 13222.31} C_VEL
LIN {X 0,Y 485.828,Z 1151.604,A -85,B 0,C 180,E1 13222.438,E2 13222.438} C_VEL
LIN {X 0,Y 485.653,Z 1156.206,A -85,B 0,C 180,E1 13226.506,E2 13226.506} C_VEL
LIN {X 0,Y 485.696,Z 1157.509,A -85,B 0,C 180,E1 13229.998,E2 13229.998} C_VEL
LIN {X 0,Y 485.728,Z 1154.51,A -85,B 0,C 180,E1 13235.368,E2 13235.368} C_VEL
LIN {X 0,Y 486.018,Z 1147.557,A -85,B 0,C 180,E1 13239.871,E2 13239.871} C_VEL
LIN {X 0,Y 487.217,Z 1134.372,A -85,B 0,C 180,E1 13244.978,E2 13244.978} C_VEL
LIN {X 0,Y 489.569,Z 1116.024,A -85,B 0,C 180,E1 13249.902,E2 13249.902} C_VEL
LIN {X 0,Y 493.759,Z 1091.805,A -85,B 0,C 180,E1 13254.713,E2 13254.713} C_VEL
LIN {X 0,Y 499.612,Z 1061.556,A -85,B 0,C 180,E1 13259.254,E2 13259.254} C_VEL
LIN {X 0,Y 506.72,Z 1026.595,A -85,B 0,C 180,E1 13263.233,E2 13263.233} C_VEL
LIN {X 0,Y 514.535,Z 986.257,A -85,B 0,C 180,E1 13266.67,E2 13266.67} C_VEL
LIN {X 0,Y 521.815,Z 942.988,A -85,B 0,C 180,E1 13269.363,E2 13269.363} C_VEL
LIN {X 0,Y 527.753,Z 899.261,A -85,B 0,C 180,E1 13271.254,E2 13271.254} C_VEL
LIN {X 0,Y 529.843,Z 872.346,A -85,B 0,C 180,E1 13272.137,E2 13272.137} C_VEL
LIN {X 0,Y 514.087,Z 836.37,A -85,B 0,C 180,E1 13274.695,E2 13274.695} C_VEL
LIN {X 0,Y 493.076,Z 799.567,A -85,B 0,C 180,E1 13277.816,E2 13277.816} C_VEL
LIN {X 0,Y 484.242,Z 784.748,A -85,B 0,C 180,E1 13279.244,E2 13279.244} C_VEL
LIN {X 0,Y 484.096,Z 783.31,A -85,B 0,C 180,E1 13279.449,E2 13279.449} C_VEL
LIN {X 0,Y 484.122,Z 783.31,A -85,B 0,C 180,E1 13285.724,E2 13285.724} C_VEL
LIN {X 0,Y 484.396,Z 783.31,A -85,B 0,C 180,E1 13292.029,E2 13292.029} C_VEL
LIN {X 0,Y 484.602,Z 783.31,A -85,B 0,C 180,E1 13297.973,E2 13297.973} C_VEL
LIN {X 0,Y 484.744,Z 783.31,A -85,B 0,C 180,E1 13303.67,E2 13303.67} C_VEL
LIN {X 0,Y 484.973,Z 783.31,A -85,B 0,C 180,E1 13309.204,E2 13309.204} C_VEL
LIN {X 0,Y 485.288,Z 783.31,A -85,B 0,C 180,E1 13314.633,E2 13314.633} C_VEL
LIN {X 0,Y 485.484,Z 783.31,A -85,B 0,C 180,E1 13320.007,E2 13320.007} C_VEL
LIN {X 0,Y 485.324,Z 783.31,A -85,B 0,C 180,E1 13325.38,E2 13325.38} C_VEL
LIN {X 0,Y 485.004,Z 783.31,A -85,B 0,C 180,E1 13330.809,E2 13330.809} C_VEL
LIN {X 0,Y 484.767,Z 783.31,A -85,B 0,C 180,E1 13336.343,E2 13336.343} C_VEL
LIN {X 0,Y 484.545,Z 783.31,A -85,B 0,C 180,E1 13342.044,E2 13342.044} C_VEL
LIN {X 0,Y 484.308,Z 783.31,A -85,B 0,C 180,E1 13347.992,E2 13347.992} C_VEL
LIN {X 0,Y 484.125,Z 783.31,A -85,B 0,C 180,E1 13354.292,E2 13354.292} C_VEL
LIN {X 0,Y 484.11,Z 783.31,A -85,B 0,C 180,E1 13358.757,E2 13358.757} C_VEL
LIN {X 0,Y 484.029,Z 783.31,A -85,B 0,C 180,E1 13363.95,E2 13363.95} C_VEL
LIN {X 0,Y 486.286,Z 788.819,A -85,B 0,C 180,E1 13364.357,E2 13364.357} C_VEL
LIN {X 0,Y 509.078,Z 826.381,A -85,B 0,C 180,E1 13367.765,E2 13367.765} C_VEL
LIN {X 0,Y 528.822,Z 866.423,A -85,B 0,C 180,E1 13370.681,E2 13370.681} C_VEL
LIN {X 0,Y 530.18,Z 872.008,A -85,B 0,C 180,E1 13370.996,E2 13370.996} C_VEL
LIN {X 0,Y 525.92,Z 912.639,A -85,B 0,C 180,E1 13372.318,E2 13372.318} C_VEL
LIN {X 0,Y 519.79,Z 953.602,A -85,B 0,C 180,E1 13374.341,E2 13374.341} C_VEL
LIN {X 0,Y 512.634,Z 991.497,A -85,B 0,C 180,E1 13376.981,E2 13376.981} C_VEL
LIN {X 0,Y 505.086,Z 1026.766,A -85,B 0,C 180,E1 13380.339,E2 13380.339} C_VEL
LIN {X 0,Y 497.922,Z 1058.719,A -85,B 0,C 180,E1 13384.456,E2 13384.456} C_VEL
LIN {X 0,Y 492.335,Z 1084.914,A -85,B 0,C 180,E1 13389.039,E2 13389.039} C_VEL
LIN {X 0,Y 488.576,Z 1105.551,A -85,B 0,C 180,E1 13394.027,E2 13394.027} C_VEL
LIN {X 0,Y 486.562,Z 1120.259,A -85,B 0,C 180,E1 13399.233,E2 13399.233} C_VEL
LIN {X 0,Y 485.867,Z 1128.039,A -85,B 0,C 180,E1 13403.735,E2 13403.735} C_VEL
LIN {X 0,Y 485.679,Z 1131.723,A -85,B 0,C 180,E1 13408.214,E2 13408.214} C_VEL
LIN {X 0,Y 485.754,Z 1131.694,A -85,B 0,C 180,E1 13411.789,E2 13411.789} C_VEL
LIN {X 0,Y 485.997,Z 1126.748,A -85,B 0,C 180,E1 13417.165,E2 13417.165} C_VEL
LIN {X 0,Y 486.946,Z 1116.829,A -85,B 0,C 180,E1 13422.093,E2 13422.093} C_VEL
LIN {X 0,Y 489.034,Z 1102.737,A -85,B 0,C 180,E1 13426.656,E2 13426.656} C_VEL
LIN {X 0,Y 492.867,Z 1082.152,A -85,B 0,C 180,E1 13431.413,E2 13431.413} C_VEL
LIN {X 0,Y 498.352,Z 1056.869,A -85,B 0,C 180,E1 13435.717,E2 13435.717} C_VEL
LIN {X 0,Y 505.274,Z 1026.05,A -85,B 0,C 180,E1 13439.638,E2 13439.638} C_VEL
LIN {X 0,Y 512.714,Z 991.015,A -85,B 0,C 180,E1 13442.959,E2 13442.959} C_VEL
LIN {X 0,Y 519.871,Z 952.219,A -85,B 0,C 180,E1 13445.656,E2 13445.656} C_VEL
LIN {X 0,Y 526.255,Z 909.867,A -85,B 0,C 180,E1 13447.699,E2 13447.699} C_VEL
LIN {X 0,Y 529.929,Z 868.947,A -85,B 0,C 180,E1 13449.03,E2 13449.03} C_VEL
LIN {X 0,Y 510.922,Z 829.749,A -85,B 0,C 180,E1 13451.87,E2 13451.87} C_VEL
LIN {X 0,Y 489.418,Z 793.811,A -85,B 0,C 180,E1 13455.037,E2 13455.037} C_VEL
LIN {X 0,Y 484.165,Z 784.708,A -85,B 0,C 180,E1 13455.89,E2 13455.89} C_VEL
LIN {X 0,Y 484.021,Z 783.31,A -85,B 0,C 180,E1 13456.055,E2 13456.055} C_VEL
LIN {X 0,Y 484.069,Z 783.31,A -85,B 0,C 180,E1 13461.494,E2 13461.494} C_VEL
LIN {X 0,Y 484.168,Z 783.31,A -85,B 0,C 180,E1 13467.855,E2 13467.855} C_VEL
LIN {X 0,Y 484.402,Z 783.31,A -85,B 0,C 180,E1 13474.025,E2 13474.025} C_VEL
LIN {X 0,Y 484.628,Z 783.31,A -85,B 0,C 180,E1 13479.88,E2 13479.88} C_VEL
LIN {X 0,Y 484.849,Z 783.31,A -85,B 0,C 180,E1 13485.646,E2 13485.646} C_VEL
LIN {X 0,Y 485.128,Z 783.31,A -85,B 0,C 180,E1 13491.01,E2 13491.01} C_VEL
LIN {X 0,Y 485.356,Z 783.31,A -85,B 0,C 180,E1 13497.422,E2 13497.422} C_VEL
LIN {X 0,Y 485.399,Z 783.31,A -85,B 0,C 180,E1 13502.689,E2 13502.689} C_VEL
LIN {X 0,Y 485.071,Z 783.31,A -85,B 0,C 180,E1 13508.978,E2 13508.978} C_VEL
LIN {X 0,Y 484.882,Z 783.31,A -85,B 0,C 180,E1 13514.468,E2 13514.468} C_VEL
LIN {X 0,Y 484.626,Z 783.31,A -85,B 0,C 180,E1 13520.288,E2 13520.288} C_VEL
LIN {X 0,Y 484.44,Z 783.31,A -85,B 0,C 180,E1 13525.958,E2 13525.958} C_VEL
LIN {X 0,Y 484.198,Z 783.31,A -85,B 0,C 180,E1 13532.337,E2 13532.337} C_VEL
LIN {X 0,Y 484.069,Z 783.31,A -85,B 0,C 180,E1 13538.744,E2 13538.744} C_VEL
LIN {X 0,Y 484.054,Z 783.504,A -85,B 0,C 180,E1 13540.725,E2 13540.725} C_VEL
LIN {X 0,Y 486.506,Z 789.037,A -85,B 0,C 180,E1 13541.161,E2 13541.161} C_VEL
LIN {X 0,Y 509.294,Z 827.574,A -85,B 0,C 180,E1 13544.624,E2 13544.624} C_VEL
LIN {X 0,Y 526.816,Z 864.217,A -85,B 0,C 180,E1 13547.309,E2 13547.309} C_VEL
LIN {X 0,Y 530.21,Z 874.703,A -85,B 0,C 180,E1 13547.987,E2 13547.987} C_VEL
LIN {X 0,Y 525.499,Z 916.636,A -85,B 0,C 180,E1 13549.416,E2 13549.416} C_VEL
LIN {X 0,Y 519.499,Z 957.279,A -85,B 0,C 180,E1 13551.432,E2 13551.432} C_VEL
LIN {X 0,Y 512.017,Z 999.366,A -85,B 0,C 180,E1 13554.341,E2 13554.341} C_VEL
LIN {X 0,Y 504.48,Z 1037.572,A -85,B 0,C 180,E1 13557.91,E2 13557.91} C_VEL
LIN {X 0,Y 497.87,Z 1070.188,A -85,B 0,C 180,E1 13561.928,E2 13561.928} C_VEL
LIN {X 0,Y 492.764,Z 1096.916,A -85,B 0,C 180,E1 13566.197,E2 13566.197} C_VEL
LIN {X 0,Y 488.969,Z 1120.04,A -85,B 0,C 180,E1 13571.035,E2 13571.035} C_VEL
LIN {X 0,Y 486.823,Z 1137.458,A -85,B 0,C 180,E1 13576.041,E2 13576.041} C_VEL
LIN {X 0,Y 485.947,Z 1149.22,A -85,B 0,C 180,E1 13581.03,E2 13581.03} C_VEL
LIN {X 0,Y 485.828,Z 1151.604,A -85,B 0,C 180,E1 13582.438,E2 13582.438} C_VEL
LIN {X 0,Y 483.283,Z 1153.716,A -85,B 0,C 180,E1 13583.938,E2 13583.938} C_VEL
LIN {X 0,Y 477.743,Z 1156.004,A -85,B 0,C 180,E1 13586.465,E2 13586.465} C_VEL
LIN {X 0,Y 477.813,Z 1157.303,A -85,B 0,C 180,E1 13589.998,E2 13589.998} C_VEL
LIN {X 0,Y 477.827,Z 1154.299,A -85,B 0,C 180,E1 13595.457,E2 13595.457} C_VEL
LIN {X 0,Y 478.145,Z 1147.334,A -85,B 0,C 180,E1 13600.035,E2 13600.035} C_VEL
LIN {X 0,Y 479.437,Z 1134.137,A -85,B 0,C 180,E1 13605.227,E2 13605.227} C_VEL
LIN {X 0,Y 481.911,Z 1115.769,A -85,B 0,C 180,E1 13610.232,E2 13610.232} C_VEL
LIN {X 0,Y 486.141,Z 1092.608,A -85,B 0,C 180,E1 13614.931,E2 13614.931} C_VEL
LIN {X 0,Y 492.17,Z 1062.88,A -85,B 0,C 180,E1 13619.508,E2 13619.508} C_VEL
LIN {X 0,Y 499.696,Z 1027.265,A -85,B 0,C 180,E1 13623.645,E2 13623.645} C_VEL
LIN {X 0,Y 507.883,Z 986.673,A -85,B 0,C 180,E1 13627.157,E2 13627.157} C_VEL
LIN {X 0,Y 515.584,Z 942.446,A -85,B 0,C 180,E1 13629.934,E2 13629.934} C_VEL
LIN {X 0,Y 521.722,Z 898.696,A -85,B 0,C 180,E1 13631.831,E2 13631.831} C_VEL
LIN {X 0,Y 523.592,Z 874.955,A -85,B 0,C 180,E1 13632.63,E2 13632.63} C_VEL
LIN {X 0,Y 508.234,Z 839.531,A -85,B 0,C 180,E1 13635.24,E2 13635.24} C_VEL
LIN {X 0,Y 486.116,Z 800.767,A -85,B 0,C 180,E1 13638.65,E2 13638.65} C_VEL
LIN {X 0,Y 476.435,Z 785.11,A -85,B 0,C 180,E1 13640.273,E2 13640.273} C_VEL
LIN {X 0,Y 476.211,Z 783.31,A -85,B 0,C 180,E1 13640.494,E2 13640.494} C_VEL
LIN {X 0,Y 476.222,Z 783.31,A -85,B 0,C 180,E1 13647.268,E2 13647.268} C_VEL
LIN {X 0,Y 476.523,Z 783.31,A -85,B 0,C 180,E1 13653.578,E2 13653.578} C_VEL
LIN {X 0,Y 476.711,Z 783.31,A -85,B 0,C 180,E1 13659.545,E2 13659.545} C_VEL
LIN {X 0,Y 476.867,Z 783.31,A -85,B 0,C 180,E1 13665.283,E2 13665.283} C_VEL
LIN {X 0,Y 477.148,Z 783.31,A -85,B 0,C 180,E1 13670.872,E2 13670.872} C_VEL
LIN {X 0,Y 477.474,Z 783.31,A -85,B 0,C 180,E1 13676.368,E2 13676.368} C_VEL
LIN {X 0,Y 477.582,Z 783.31,A -85,B 0,C 180,E1 13681.825,E2 13681.825} C_VEL
LIN {X 0,Y 477.252,Z 783.31,A -85,B 0,C 180,E1 13687.302,E2 13687.302} C_VEL
LIN {X 0,Y 476.993,Z 783.31,A -85,B 0,C 180,E1 13692.853,E2 13692.853} C_VEL
LIN {X 0,Y 476.735,Z 783.31,A -85,B 0,C 180,E1 13698.537,E2 13698.537} C_VEL
LIN {X 0,Y 476.493,Z 783.31,A -85,B 0,C 180,E1 13704.422,E2 13704.422} C_VEL
LIN {X 0,Y 476.269,Z 783.31,A -85,B 0,C 180,E1 13710.804,E2 13710.804} C_VEL
LIN {X 0,Y 476.121,Z 783.31,A -85,B 0,C 180,E1 13717.293,E2 13717.293} C_VEL
LIN {X 0,Y 476.066,Z 783.311,A -85,B 0,C 180,E1 13722.887,E2 13722.887} C_VEL
LIN {X 0,Y 478.482,Z 788.954,A -85,B 0,C 180,E1 13723.337,E2 13723.337} C_VEL
LIN {X 0,Y 501.602,Z 826.642,A -85,B 0,C 180,E1 13726.942,E2 13726.942} C_VEL
LIN {X 0,Y 521.376,Z 866.316,A -85,B 0,C 180,E1 13729.962,E2 13729.962} C_VEL
LIN {X 0,Y 523.973,Z 874.501,A -85,B 0,C 180,E1 13730.495,E2 13730.495} C_VEL
LIN {X 0,Y 519.328,Z 915.69,A -85,B 0,C 180,E1 13731.888,E2 13731.888} C_VEL
LIN {X 0,Y 513.388,Z 954.045,A -85,B 0,C 180,E1 13733.826,E2 13733.826} C_VEL
LIN {X 0,Y 505.975,Z 991.871,A -85,B 0,C 180,E1 13736.489,E2 13736.489} C_VEL
LIN {X 0,Y 498.043,Z 1027.586,A -85,B 0,C 180,E1 13739.94,E2 13739.94} C_VEL
LIN {X 0,Y 490.588,Z 1059.307,A -85,B 0,C 180,E1 13744.1,E2 13744.1} C_VEL
LIN {X 0,Y 484.828,Z 1085.162,A -85,B 0,C 180,E1 13748.699,E2 13748.699} C_VEL
LIN {X 0,Y 481.013,Z 1105.012,A -85,B 0,C 180,E1 13753.533,E2 13753.533} C_VEL
LIN {X 0,Y 478.775,Z 1120.006,A -85,B 0,C 180,E1 13758.835,E2 13758.835} C_VEL
LIN {X 0,Y 478.002,Z 1128.25,A -85,B 0,C 180,E1 13763.632,E2 13763.632} C_VEL
LIN {X 0,Y 477.785,Z 1131.93,A -85,B 0,C 180,E1 13768.184,E2 13768.184} C_VEL
LIN {X 0,Y 477.857,Z 1131.901,A -85,B 0,C 180,E1 13771.819,E2 13771.819} C_VEL
LIN {X 0,Y 478.117,Z 1126.962,A -85,B 0,C 180,E1 13777.284,E2 13777.284} C_VEL
LIN {X 0,Y 479.149,Z 1116.936,A -85,B 0,C 180,E1 13782.341,E2 13782.341} C_VEL
LIN {X 0,Y 481.6,Z 1101.292,A -85,B 0,C 180,E1 13787.392,E2 13787.392} C_VEL
LIN {X 0,Y 485.611,Z 1081.241,A -85,B 0,C 180,E1 13791.99,E2 13791.99} C_VEL
LIN {X 0,Y 491.464,Z 1055.433,A -85,B 0,C 180,E1 13796.376,E2 13796.376} C_VEL
LIN {X 0,Y 498.618,Z 1025.007,A -85,B 0,C 180,E1 13800.241,E2 13800.241} C_VEL
LIN {X 0,Y 506.179,Z 990.781,A -85,B 0,C 180,E1 13803.499,E2 13803.499} C_VEL
LIN {X 0,Y 513.471,Z 952.708,A -85,B 0,C 180,E1 13806.17,E2 13806.17} C_VEL
LIN {X 0,Y 520.123,Z 910.092,A -85,B 0,C 180,E1 13808.246,E2 13808.246} C_VEL
LIN {X 0,Y 523.726,Z 871.864,A -85,B 0,C 180,E1 13809.518,E2 13809.518} C_VEL
LIN {X 0,Y 505.708,Z 833.983,A -85,B 0,C 180,E1 13812.357,E2 13812.357} C_VEL
LIN {X 0,Y 482.54,Z 795.086,A -85,B 0,C 180,E1 13815.886,E2 13815.886} C_VEL
LIN {X 0,Y 476.214,Z 784.795,A -85,B 0,C 180,E1 13816.947,E2 13816.947} C_VEL
LIN {X 0,Y 476.055,Z 783.31,A -85,B 0,C 180,E1 13817.059,E2 13817.059} C_VEL
LIN {X 0,Y 476.083,Z 783.31,A -85,B 0,C 180,E1 13822.789,E2 13822.789} C_VEL
LIN {X 0,Y 476.295,Z 783.31,A -85,B 0,C 180,E1 13829.399,E2 13829.399} C_VEL
LIN {X 0,Y 476.537,Z 783.31,A -85,B 0,C 180,E1 13835.58,E2 13835.58} C_VEL
LIN {X 0,Y 476.754,Z 783.31,A -85,B 0,C 180,E1 13841.464,E2 13841.464} C_VEL
LIN {X 0,Y 476.97,Z 783.31,A -85,B 0,C 180,E1 13847.146,E2 13847.146} C_VEL
LIN {X 0,Y 477.295,Z 783.31,A -85,B 0,C 180,E1 13852.699,E2 13852.699} C_VEL
LIN {X 0,Y 477.527,Z 783.31,A -85,B 0,C 180,E1 13858.175,E2 13858.175} C_VEL
LIN {X 0,Y 477.476,Z 783.31,A -85,B 0,C 180,E1 13863.632,E2 13863.632} C_VEL
LIN {X 0,Y 477.081,Z 783.31,A -85,B 0,C 180,E1 13870.083,E2 13870.083} C_VEL
LIN {X 0,Y 476.866,Z 783.31,A -85,B 0,C 180,E1 13876.608,E2 13876.608} C_VEL
LIN {X 0,Y 476.584,Z 783.31,A -85,B 0,C 180,E1 13882.78,E2 13882.78} C_VEL
LIN {X 0,Y 476.449,Z 783.31,A -85,B 0,C 180,E1 13888.48,E2 13888.48} C_VEL
LIN {X 0,Y 476.195,Z 783.31,A -85,B 0,C 180,E1 13894.928,E2 13894.928} C_VEL
LIN {X 0,Y 476.169,Z 783.31,A -85,B 0,C 180,E1 13899.668,E2 13899.668} C_VEL
LIN {X 0,Y 478.536,Z 788.965,A -85,B 0,C 180,E1 13900.122,E2 13900.122} C_VEL
LIN {X 0,Y 501.649,Z 827.297,A -85,B 0,C 180,E1 13903.779,E2 13903.779} C_VEL
LIN {X 0,Y 519.907,Z 865.131,A -85,B 0,C 180,E1 13906.676,E2 13906.676} C_VEL
LIN {X 0,Y 523.922,Z 878.047,A -85,B 0,C 180,E1 13907.52,E2 13907.52} C_VEL
LIN {X 0,Y 518.671,Z 920.917,A -85,B 0,C 180,E1 13909.045,E2 13909.045} C_VEL
LIN {X 0,Y 512.613,Z 960.339,A -85,B 0,C 180,E1 13911.088,E2 13911.088} C_VEL
LIN {X 0,Y 505.119,Z 1000.606,A -85,B 0,C 180,E1 13913.934,E2 13913.934} C_VEL
LIN {X 0,Y 497.166,Z 1039.367,A -85,B 0,C 180,E1 13917.638,E2 13917.638} C_VEL
LIN {X 0,Y 489.91,Z 1073.429,A -85,B 0,C 180,E1 13921.975,E2 13921.975} C_VEL
LIN {X 0,Y 484.215,Z 1102.717,A -85,B 0,C 180,E1 13926.952,E2 13926.952} C_VEL
LIN {X 0,Y 480.486,Z 1125.071,A -85,B 0,C 180,E1 13932.092,E2 13932.092} C_VEL
LIN {X 0,Y 478.656,Z 1140.952,A -85,B 0,C 180,E1 13937.196,E2 13937.196} C_VEL
LIN {X 0,Y 477.973,Z 1150.621,A -85,B 0,C 180,E1 13941.797,E2 13941.797} C_VEL
LIN {X 0,Y 477.743,Z 1156.004,A -85,B 0,C 180,E1 13946.465,E2 13946.465} C_VEL
LIN {X 0,Y 473.78,Z 1156.915,A -85,B 0,C 180,E1 13948.51,E2 13948.51} C_VEL
LIN {X 0,Y 469.839,Z 1156.983,A -85,B 0,C 180,E1 13950.59,E2 13950.59} C_VEL
LIN {X 0,Y 469.941,Z 1154.089,A -85,B 0,C 180,E1 13955.549,E2 13955.549} C_VEL
LIN {X 0,Y 470.339,Z 1146.224,A -85,B 0,C 180,E1 13960.622,E2 13960.622} C_VEL
LIN {X 0,Y 471.856,Z 1132.124,A -85,B 0,C 180,E1 13966.077,E2 13966.077} C_VEL
LIN {X 0,Y 475.152,Z 1111.507,A -85,B 0,C 180,E1 13971.511,E2 13971.511} C_VEL
LIN {X 0,Y 480.388,Z 1084.448,A -85,B 0,C 180,E1 13976.707,E2 13976.707} C_VEL
LIN {X 0,Y 487.517,Z 1051.411,A -85,B 0,C 180,E1 13981.429,E2 13981.429} C_VEL
LIN {X 0,Y 495.612,Z 1014.593,A -85,B 0,C 180,E1 13985.361,E2 13985.361} C_VEL
LIN {X 0,Y 503.629,Z 974.533,A -85,B 0,C 180,E1 13988.554,E2 13988.554} C_VEL
LIN {X 0,Y 510.875,Z 932.164,A -85,B 0,C 180,E1 13991.008,E2 13991.008} C_VEL
LIN {X 0,Y 516.738,Z 889.011,A -85,B 0,C 180,E1 13992.728,E2 13992.728} C_VEL
LIN {X 0,Y 517.214,Z 877.132,A -85,B 0,C 180,E1 13993.168,E2 13993.168} C_VEL
